LIN {X 0,Y 136.247,Z 303.137,A -85,B 0,C 180,E1 -24818.833,E2 -24818.833} C_VEL
LIN {X 0,Y 136.271,Z 303.129,A -85,B 0,C 180,E1 -24825.056,E2 -24825.056} C_VEL
LIN {X 0,Y 136.434,Z 303.114,A -85,B 0,C 180,E1 -24828.164,E2 -24828.164} C_VEL
LIN {X 0,Y 136.551,Z 303.099,A -85,B 0,C 180,E1 -24831.117,E2 -24831.117} C_VEL
LIN {X 0,Y 137.132,Z 303.026,A -85,B 0,C 180,E1 -24839.999,E2 -24839.999} C_VEL
LIN {X 0,Y 136.551,Z 303.097,A -85,B 0,C 180,E1 -24848.882,E2 -24848.882} C_VEL
LIN {X 0,Y 136.442,Z 303.112,A -85,B 0,C 180,E1 -24851.889,E2 -24851.889} C_VEL
LIN {X 0,Y 136.252,Z 303.133,A -85,B 0,C 180,E1 -24858.027,E2 -24858.027} C_VEL
LIN {X 0,Y 136.434,Z 303.14,A -85,B 0,C 180,E1 -24864.336,E2 -24864.336} C_VEL
LIN {X 0,Y 136.755,Z 306.874,A -85,B 0,C 180,E1 -24870.924,E2 -24870.924} C_VEL
LIN {X 0,Y 137.423,Z 309.535,A -85,B 0,C 180,E1 -24875.456,E2 -24875.456} C_VEL
LIN {X 0,Y 143.688,Z 330.399,A -85,B 0,C 180,E1 -24879.825,E2 -24879.825} C_VEL
LIN {X 0,Y 145.662,Z 339.16,A -85,B 0,C 180,E1 -24881.689,E2 -24881.689} C_VEL
LIN {X 0,Y 147.43,Z 355.491,A -85,B 0,C 180,E1 -24885.229,E2 -24885.229} C_VEL
LIN {X 0,Y 148.861,Z 369.384,A -85,B 0,C 180,E1 -24888.626,E2 -24888.626} C_VEL
LIN {X 0,Y 150.113,Z 381.659,A -85,B 0,C 180,E1 -24891.987,E2 -24891.987} C_VEL
LIN {X 0,Y 150.686,Z 388.239,A -85,B 0,C 180,E1 -24893.945,E2 -24893.945} C_VEL
LIN {X 0,Y 146.918,Z 399.34,A -85,B 0,C 180,E1 -24897.441,E2 -24897.441} C_VEL
LIN {X 0,Y 142.825,Z 411.303,A -85,B 0,C 180,E1 -24902.116,E2 -24902.116} C_VEL
LIN {X 0,Y 139.666,Z 421.52,A -85,B 0,C 180,E1 -24907.046,E2 -24907.046} C_VEL
LIN {X 0,Y 137.366,Z 430.082,A -85,B 0,C 180,E1 -24912.123,E2 -24912.123} C_VEL
LIN {X 0,Y 135.876,Z 438.21,A -85,B 0,C 180,E1 -24918.059,E2 -24918.059} C_VEL
LIN {X 0,Y 135.342,Z 444.688,A -85,B 0,C 180,E1 -24924.039,E2 -24924.039} C_VEL
LIN {X 0,Y 135.239,Z 448.491,A -85,B 0,C 180,E1 -24928.511,E2 -24928.511} C_VEL
LIN {X 0,Y 135.256,Z 449.575,A -85,B 0,C 180,E1 -24930,E2 -24930} C_VEL
LIN {X 0,Y 135.01,Z 451.418,A -85,B 0,C 180,E1 -24932.984,E2 -24932.984} C_VEL
LIN {X 0,Y 134.714,Z 453.637,A -85,B 0,C 180,E1 -24937.6,E2 -24937.6} C_VEL
LIN {X 0,Y 135.394,Z 456.033,A -85,B 0,C 180,E1 -24945.043,E2 -24945.043} C_VEL
LIN {X 0,Y 139.13,Z 457.397,A -85,B 0,C 180,E1 -24953.835,E2 -24953.835} C_VEL
LIN {X 0,Y 146.373,Z 457.366,A -85,B 0,C 180,E1 -24961.881,E2 -24961.881} C_VEL
LIN {X 0,Y 156.505,Z 456.017,A -85,B 0,C 180,E1 -24968.953,E2 -24968.953} C_VEL
LIN {X 0,Y 164.765,Z 454.523,A -85,B 0,C 180,E1 -24973.038,E2 -24973.038} C_VEL
LIN {X 0,Y 169.344,Z 453.57,A -85,B 0,C 180,E1 -24974.872,E2 -24974.872} C_VEL
LIN {X 0,Y 170.849,Z 453.204,A -85,B 0,C 180,E1 -24975.629,E2 -24975.629} C_VEL
LIN {X 0,Y 158.161,Z 452.885,A -85,B 0,C 180,E1 -24981.531,E2 -24981.531} C_VEL
LIN {X 0,Y 150.957,Z 451.853,A -85,B 0,C 180,E1 -24986.036,E2 -24986.036} C_VEL
LIN {X 0,Y 144.974,Z 450.016,A -85,B 0,C 180,E1 -24991.003,E2 -24991.003} C_VEL
LIN {X 0,Y 140.598,Z 447.636,A -85,B 0,C 180,E1 -24995.993,E2 -24995.993} C_VEL
LIN {X 0,Y 138.42,Z 446.349,A -85,B 0,C 180,E1 -24998.183,E2 -24998.183} C_VEL
LIN {X 0,Y 133.615,Z 443.7,A -85,B 0,C 180,E1 -25001.66,E2 -25001.66} C_VEL
LIN {X 0,Y 130.02,Z 441.226,A -85,B 0,C 180,E1 -25004.557,E2 -25004.557} C_VEL
LIN {X 0,Y 128.29,Z 439.216,A -85,B 0,C 180,E1 -25006.914,E2 -25006.914} C_VEL
LIN {X 0,Y 128.014,Z 438.527,A -85,B 0,C 180,E1 -25007.737,E2 -25007.737} C_VEL
LIN {X 0,Y 127.224,Z 432.975,A -85,B 0,C 180,E1 -25013.906,E2 -25013.906} C_VEL
LIN {X 0,Y 127.191,Z 428.154,A -85,B 0,C 180,E1 -25018.418,E2 -25018.418} C_VEL
LIN {X 0,Y 127.646,Z 420.139,A -85,B 0,C 180,E1 -25024.738,E2 -25024.738} C_VEL
LIN {X 0,Y 128.792,Z 410.762,A -85,B 0,C 180,E1 -25030.813,E2 -25030.813} C_VEL
LIN {X 0,Y 131.133,Z 398.794,A -85,B 0,C 180,E1 -25037.144,E2 -25037.144} C_VEL
LIN {X 0,Y 133.545,Z 388.569,A -85,B 0,C 180,E1 -25041.617,E2 -25041.617} C_VEL
LIN {X 0,Y 137.26,Z 374.549,A -85,B 0,C 180,E1 -25046.617,E2 -25046.617} C_VEL
LIN {X 0,Y 140.984,Z 360.329,A -85,B 0,C 180,E1 -25050.729,E2 -25050.729} C_VEL
LIN {X 0,Y 143.252,Z 351.164,A -85,B 0,C 180,E1 -25052.95,E2 -25052.95} C_VEL
LIN {X 0,Y 140.82,Z 340.487,A -85,B 0,C 180,E1 -25055.806,E2 -25055.806} C_VEL
LIN {X 0,Y 136.648,Z 326.02,A -85,B 0,C 180,E1 -25059.514,E2 -25059.514} C_VEL
LIN {X 0,Y 131.962,Z 312.426,A -85,B 0,C 180,E1 -25062.921,E2 -25062.921} C_VEL
LIN {X 0,Y 128.958,Z 304.05,A -85,B 0,C 180,E1 -25065.024,E2 -25065.024} C_VEL
LIN {X 0,Y 128.938,Z 304.048,A -85,B 0,C 180,E1 -25069.739,E2 -25069.739} C_VEL
LIN {X 0,Y 128.983,Z 304.045,A -85,B 0,C 180,E1 -25074.819,E2 -25074.819} C_VEL
LIN {X 0,Y 129.019,Z 304.038,A -85,B 0,C 180,E1 -25080.643,E2 -25080.643} C_VEL
LIN {X 0,Y 129.033,Z 304.037,A -85,B 0,C 180,E1 -25084.168,E2 -25084.168} C_VEL
LIN {X 0,Y 129.11,Z 304.023,A -85,B 0,C 180,E1 -25087.728,E2 -25087.728} C_VEL
LIN {X 0,Y 129.156,Z 304.021,A -85,B 0,C 180,E1 -25090.944,E2 -25090.944} C_VEL
LIN {X 0,Y 129.392,Z 303.991,A -85,B 0,C 180,E1 -25097.876,E2 -25097.876} C_VEL
LIN {X 0,Y 129.475,Z 303.98,A -85,B 0,C 180,E1 -25100.628,E2 -25100.628} C_VEL
LIN {X 0,Y 130.087,Z 303.902,A -85,B 0,C 180,E1 -25110,E2 -25110} C_VEL
LIN {X 0,Y 129.481,Z 303.976,A -85,B 0,C 180,E1 -25119.372,E2 -25119.372} C_VEL
LIN {X 0,Y 129.355,Z 303.996,A -85,B 0,C 180,E1 -25122.552,E2 -25122.552} C_VEL
LIN {X 0,Y 129.187,Z 304.013,A -85,B 0,C 180,E1 -25129.051,E2 -25129.051} C_VEL
LIN {X 0,Y 129.139,Z 304.023,A -85,B 0,C 180,E1 -25132.393,E2 -25132.393} C_VEL
LIN {X 0,Y 129.038,Z 304.037,A -85,B 0,C 180,E1 -25139.373,E2 -25139.373} C_VEL
LIN {X 0,Y 128.959,Z 304.041,A -85,B 0,C 180,E1 -25145.167,E2 -25145.167} C_VEL
LIN {X 0,Y 128.924,Z 304.048,A -85,B 0,C 180,E1 -25150.856,E2 -25150.856} C_VEL
LIN {X 0,Y 128.914,Z 304.052,A -85,B 0,C 180,E1 -25155.132,E2 -25155.132} C_VEL
LIN {X 0,Y 128.938,Z 304.044,A -85,B 0,C 180,E1 -25159.739,E2 -25159.739} C_VEL
LIN {X 0,Y 128.983,Z 304.044,A -85,B 0,C 180,E1 -25164.818,E2 -25164.818} C_VEL
LIN {X 0,Y 129.019,Z 304.036,A -85,B 0,C 180,E1 -25170.642,E2 -25170.642} C_VEL
LIN {X 0,Y 129.033,Z 304.037,A -85,B 0,C 180,E1 -25174.167,E2 -25174.167} C_VEL
LIN {X 0,Y 129.11,Z 304.021,A -85,B 0,C 180,E1 -25177.727,E2 -25177.727} C_VEL
LIN {X 0,Y 129.156,Z 304.022,A -85,B 0,C 180,E1 -25180.943,E2 -25180.943} C_VEL
LIN {X 0,Y 129.392,Z 303.99,A -85,B 0,C 180,E1 -25187.875,E2 -25187.875} C_VEL
LIN {X 0,Y 129.475,Z 303.981,A -85,B 0,C 180,E1 -25190.627,E2 -25190.627} C_VEL
LIN {X 0,Y 130.087,Z 303.904,A -85,B 0,C 180,E1 -25199.999,E2 -25199.999} C_VEL
LIN {X 0,Y 129.477,Z 303.978,A -85,B 0,C 180,E1 -25209.371,E2 -25209.371} C_VEL
LIN {X 0,Y 129.346,Z 303.996,A -85,B 0,C 180,E1 -25212.552,E2 -25212.552} C_VEL
LIN {X 0,Y 129.179,Z 304.015,A -85,B 0,C 180,E1 -25219.052,E2 -25219.052} C_VEL
LIN {X 0,Y 129.367,Z 304.154,A -85,B 0,C 180,E1 -25224.898,E2 -25224.898} C_VEL
LIN {X 0,Y 129.882,Z 308.439,A -85,B 0,C 180,E1 -25232.758,E2 -25232.758} C_VEL
LIN {X 0,Y 130.109,Z 309.14,A -85,B 0,C 180,E1 -25233.967,E2 -25233.967} C_VEL
LIN {X 0,Y 136.026,Z 328.806,A -85,B 0,C 180,E1 -25238.315,E2 -25238.315} C_VEL
LIN {X 0,Y 138.682,Z 339.25,A -85,B 0,C 180,E1 -25240.718,E2 -25240.718} C_VEL
LIN {X 0,Y 140.292,Z 353.804,A -85,B 0,C 180,E1 -25244.032,E2 -25244.032} C_VEL
LIN {X 0,Y 141.788,Z 369.4,A -85,B 0,C 180,E1 -25248.03,E2 -25248.03} C_VEL
LIN {X 0,Y 143.073,Z 382.421,A -85,B 0,C 180,E1 -25251.807,E2 -25251.807} C_VEL
LIN {X 0,Y 143.609,Z 387.897,A -85,B 0,C 180,E1 -25253.526,E2 -25253.526} C_VEL
LIN {X 0,Y 139.712,Z 399.089,A -85,B 0,C 180,E1 -25257.264,E2 -25257.264} C_VEL
LIN {X 0,Y 135.93,Z 409.933,A -85,B 0,C 180,E1 -25261.706,E2 -25261.706} C_VEL
LIN {X 0,Y 132.843,Z 419.722,A -85,B 0,C 180,E1 -25266.622,E2 -25266.622} C_VEL
LIN {X 0,Y 130.472,Z 428.371,A -85,B 0,C 180,E1 -25271.957,E2 -25271.957} C_VEL
LIN {X 0,Y 129.087,Z 435.667,A -85,B 0,C 180,E1 -25277.421,E2 -25277.421} C_VEL
LIN {X 0,Y 128.494,Z 442.455,A -85,B 0,C 180,E1 -25283.72,E2 -25283.72} C_VEL
LIN {X 0,Y 128.382,Z 446.483,A -85,B 0,C 180,E1 -25288.431,E2 -25288.431} C_VEL
LIN {X 0,Y 128.387,Z 447.654,A -85,B 0,C 180,E1 -25290,E2 -25290} C_VEL
LIN {X 0,Y 128.146,Z 449.612,A -85,B 0,C 180,E1 -25293.144,E2 -25293.144} C_VEL
LIN {X 0,Y 127.839,Z 452.095,A -85,B 0,C 180,E1 -25298.294,E2 -25298.294} C_VEL
LIN {X 0,Y 128.636,Z 454.561,A -85,B 0,C 180,E1 -25305.853,E2 -25305.853} C_VEL
LIN {X 0,Y 132.681,Z 456.227,A -85,B 0,C 180,E1 -25315.072,E2 -25315.072} C_VEL
LIN {X 0,Y 140.385,Z 456.546,A -85,B 0,C 180,E1 -25323.414,E2 -25323.414} C_VEL
LIN {X 0,Y 151.043,Z 455.659,A -85,B 0,C 180,E1 -25330.649,E2 -25330.649} C_VEL
LIN {X 0,Y 159.649,Z 454.433,A -85,B 0,C 180,E1 -25334.777,E2 -25334.777} C_VEL
LIN {X 0,Y 161.243,Z 454.077,A -85,B 0,C 180,E1 -25335.783,E2 -25335.783} C_VEL
LIN {X 0,Y 152.661,Z 453.441,A -85,B 0,C 180,E1 -25339.872,E2 -25339.872} C_VEL
LIN {X 0,Y 141.781,Z 451.137,A -85,B 0,C 180,E1 -25346.958,E2 -25346.958} C_VEL
LIN {X 0,Y 136.124,Z 448.673,A -85,B 0,C 180,E1 -25352.312,E2 -25352.312} C_VEL
LIN {X 0,Y 131.776,Z 445.435,A -85,B 0,C 180,E1 -25358.08,E2 -25358.08} C_VEL
LIN {X 0,Y 128.491,Z 440.128,A -85,B 0,C 180,E1 -25365.752,E2 -25365.752} C_VEL
LIN {X 0,Y 128.014,Z 438.527,A -85,B 0,C 180,E1 -25367.737,E2 -25367.737} C_VEL
LIN {X 0,Y 126.912,Z 436.36,A -85,B 0,C 180,E1 -25370.152,E2 -25370.152} C_VEL
LIN {X 0,Y 125.08,Z 433.957,A -85,B 0,C 180,E1 -25372.473,E2 -25372.473} C_VEL
LIN {X 0,Y 121.241,Z 428.484,A -85,B 0,C 180,E1 -25377.122,E2 -25377.122} C_VEL
LIN {X 0,Y 120.269,Z 425.573,A -85,B 0,C 180,E1 -25379.558,E2 -25379.558} C_VEL
LIN {X 0,Y 120.223,Z 424.572,A -85,B 0,C 180,E1 -25380.384,E2 -25380.384} C_VEL
LIN {X 0,Y 120.757,Z 417.504,A -85,B 0,C 180,E1 -25385.846,E2 -25385.846} C_VEL
LIN {X 0,Y 122.135,Z 407.431,A -85,B 0,C 180,E1 -25392.378,E2 -25392.378} C_VEL
LIN {X 0,Y 124.432,Z 396.651,A -85,B 0,C 180,E1 -25398.099,E2 -25398.099} C_VEL
LIN {X 0,Y 127.486,Z 384.124,A -85,B 0,C 180,E1 -25403.559,E2 -25403.559} C_VEL
LIN {X 0,Y 130.911,Z 371.667,A -85,B 0,C 180,E1 -25408.019,E2 -25408.019} C_VEL
LIN {X 0,Y 134.564,Z 358.197,A -85,B 0,C 180,E1 -25411.921,E2 -25411.921} C_VEL
LIN {X 0,Y 136.065,Z 352.541,A -85,B 0,C 180,E1 -25413.345,E2 -25413.345} C_VEL
LIN {X 0,Y 135.805,Z 349.78,A -85,B 0,C 180,E1 -25414.104,E2 -25414.104} C_VEL
LIN {X 0,Y 132.825,Z 337.831,A -85,B 0,C 180,E1 -25417.469,E2 -25417.469} C_VEL
LIN {X 0,Y 128.684,Z 324.087,A -85,B 0,C 180,E1 -25421.208,E2 -25421.208} C_VEL
LIN {X 0,Y 123.585,Z 309.815,A -85,B 0,C 180,E1 -25424.977,E2 -25424.977} C_VEL
LIN {X 0,Y 121.846,Z 304.934,A -85,B 0,C 180,E1 -25426.367,E2 -25426.367} C_VEL
LIN {X 0,Y 121.858,Z 304.931,A -85,B 0,C 180,E1 -25430.623,E2 -25430.623} C_VEL
LIN {X 0,Y 121.935,Z 304.922,A -85,B 0,C 180,E1 -25434.804,E2 -25434.804} C_VEL
LIN {X 0,Y 121.931,Z 304.921,A -85,B 0,C 180,E1 -25439.837,E2 -25439.837} C_VEL
LIN {X 0,Y 121.986,Z 304.909,A -85,B 0,C 180,E1 -25446.216,E2 -25446.216} C_VEL
LIN {X 0,Y 122.048,Z 304.906,A -85,B 0,C 180,E1 -25449.787,E2 -25449.787} C_VEL
LIN {X 0,Y 122.242,Z 304.882,A -85,B 0,C 180,E1 -25456.705,E2 -25456.705} C_VEL
LIN {X 0,Y 122.411,Z 304.862,A -85,B 0,C 180,E1 -25460.082,E2 -25460.082} C_VEL
LIN {X 0,Y 122.591,Z 304.839,A -85,B 0,C 180,E1 -25466.714,E2 -25466.714} C_VEL
LIN {X 0,Y 123.04,Z 304.779,A -85,B 0,C 180,E1 -25470,E2 -25470} C_VEL
LIN {X 0,Y 122.424,Z 304.859,A -85,B 0,C 180,E1 -25476.593,E2 -25476.593} C_VEL
LIN {X 0,Y 122.417,Z 304.856,A -85,B 0,C 180,E1 -25479.918,E2 -25479.918} C_VEL
LIN {X 0,Y 122.249,Z 304.882,A -85,B 0,C 180,E1 -25483.295,E2 -25483.295} C_VEL
LIN {X 0,Y 122.076,Z 304.903,A -85,B 0,C 180,E1 -25490.208,E2 -25490.208} C_VEL
LIN {X 0,Y 121.999,Z 304.911,A -85,B 0,C 180,E1 -25493.782,E2 -25493.782} C_VEL
LIN {X 0,Y 121.942,Z 304.92,A -85,B 0,C 180,E1 -25500.171,E2 -25500.171} C_VEL
LIN {X 0,Y 121.883,Z 304.925,A -85,B 0,C 180,E1 -25506.169,E2 -25506.169} C_VEL
LIN {X 0,Y 121.865,Z 304.925,A -85,B 0,C 180,E1 -25511.433,E2 -25511.433} C_VEL
LIN {X 0,Y 121.866,Z 304.929,A -85,B 0,C 180,E1 -25518.566,E2 -25518.566} C_VEL
LIN {X 0,Y 121.935,Z 304.922,A -85,B 0,C 180,E1 -25524.803,E2 -25524.803} C_VEL
LIN {X 0,Y 121.931,Z 304.916,A -85,B 0,C 180,E1 -25529.836,E2 -25529.836} C_VEL
LIN {X 0,Y 121.986,Z 304.91,A -85,B 0,C 180,E1 -25536.215,E2 -25536.215} C_VEL
LIN {X 0,Y 122.048,Z 304.905,A -85,B 0,C 180,E1 -25539.787,E2 -25539.787} C_VEL
LIN {X 0,Y 122.242,Z 304.879,A -85,B 0,C 180,E1 -25546.704,E2 -25546.704} C_VEL
LIN {X 0,Y 122.411,Z 304.863,A -85,B 0,C 180,E1 -25550.081,E2 -25550.081} C_VEL
LIN {X 0,Y 122.594,Z 304.839,A -85,B 0,C 180,E1 -25556.713,E2 -25556.713} C_VEL
LIN {X 0,Y 123.041,Z 304.781,A -85,B 0,C 180,E1 -25559.999,E2 -25559.999} C_VEL
LIN {X 0,Y 122.423,Z 304.86,A -85,B 0,C 180,E1 -25566.592,E2 -25566.592} C_VEL
LIN {X 0,Y 122.407,Z 304.857,A -85,B 0,C 180,E1 -25569.918,E2 -25569.918} C_VEL
LIN {X 0,Y 122.242,Z 304.882,A -85,B 0,C 180,E1 -25573.295,E2 -25573.295} C_VEL
LIN {X 0,Y 122.118,Z 304.899,A -85,B 0,C 180,E1 -25580.2,E2 -25580.2} C_VEL
LIN {X 0,Y 122.314,Z 304.914,A -85,B 0,C 180,E1 -25585.071,E2 -25585.071} C_VEL
LIN {X 0,Y 122.754,Z 308.868,A -85,B 0,C 180,E1 -25592.34,E2 -25592.34} C_VEL
LIN {X 0,Y 127.805,Z 325.454,A -85,B 0,C 180,E1 -25596.272,E2 -25596.272} C_VEL
LIN {X 0,Y 131.407,Z 338.28,A -85,B 0,C 180,E1 -25599.427,E2 -25599.427} C_VEL
LIN {X 0,Y 132.448,Z 344.471,A -85,B 0,C 180,E1 -25600.907,E2 -25600.907} C_VEL
LIN {X 0,Y 133.798,Z 359.38,A -85,B 0,C 180,E1 -25604.631,E2 -25604.631} C_VEL
LIN {X 0,Y 135.224,Z 374.386,A -85,B 0,C 180,E1 -25608.901,E2 -25608.901} C_VEL
LIN {X 0,Y 136.456,Z 387.871,A -85,B 0,C 180,E1 -25613.221,E2 -25613.221} C_VEL
LIN {X 0,Y 131.894,Z 400.51,A -85,B 0,C 180,E1 -25617.801,E2 -25617.801} C_VEL
LIN {X 0,Y 127.911,Z 412.021,A -85,B 0,C 180,E1 -25623.045,E2 -25623.045} C_VEL
LIN {X 0,Y 124.607,Z 423.026,A -85,B 0,C 180,E1 -25629.359,E2 -25629.359} C_VEL
LIN {X 0,Y 122.525,Z 432.013,A -85,B 0,C 180,E1 -25635.89,E2 -25635.89} C_VEL
LIN {X 0,Y 121.753,Z 438.493,A -85,B 0,C 180,E1 -25641.703,E2 -25641.703} C_VEL
LIN {X 0,Y 121.596,Z 443.062,A -85,B 0,C 180,E1 -25646.686,E2 -25646.686} C_VEL
LIN {X 0,Y 121.575,Z 445.568,A -85,B 0,C 180,E1 -25650,E2 -25650} C_VEL
LIN {X 0,Y 121.339,Z 447.639,A -85,B 0,C 180,E1 -25653.32,E2 -25653.32} C_VEL
LIN {X 0,Y 121.022,Z 450.427,A -85,B 0,C 180,E1 -25659.174,E2 -25659.174} C_VEL
LIN {X 0,Y 121.921,Z 452.992,A -85,B 0,C 180,E1 -25666.751,E2 -25666.751} C_VEL
LIN {X 0,Y 126.339,Z 454.977,A -85,B 0,C 180,E1 -25676.425,E2 -25676.425} C_VEL
LIN {X 0,Y 134.514,Z 455.608,A -85,B 0,C 180,E1 -25685.08,E2 -25685.08} C_VEL
LIN {X 0,Y 145.726,Z 455.082,A -85,B 0,C 180,E1 -25692.469,E2 -25692.469} C_VEL
LIN {X 0,Y 150.039,Z 454.695,A -85,B 0,C 180,E1 -25694.638,E2 -25694.638} C_VEL
LIN {X 0,Y 151.661,Z 454.387,A -85,B 0,C 180,E1 -25695.965,E2 -25695.965} C_VEL
LIN {X 0,Y 139.375,Z 452.212,A -85,B 0,C 180,E1 -25702.765,E2 -25702.765} C_VEL
LIN {X 0,Y 129.857,Z 448.425,A -85,B 0,C 180,E1 -25710.851,E2 -25710.851} C_VEL
LIN {X 0,Y 124.324,Z 443.944,A -85,B 0,C 180,E1 -25718.443,E2 -25718.443} C_VEL
LIN {X 0,Y 121.217,Z 438.065,A -85,B 0,C 180,E1 -25726.591,E2 -25726.591} C_VEL
LIN {X 0,Y 120.196,Z 431.125,A -85,B 0,C 180,E1 -25734.391,E2 -25734.391} C_VEL
LIN {X 0,Y 120.223,Z 424.572,A -85,B 0,C 180,E1 -25740.384,E2 -25740.384} C_VEL
LIN {X 0,Y 119.727,Z 421.513,A -85,B 0,C 180,E1 -25742.772,E2 -25742.772} C_VEL
LIN {X 0,Y 117.359,Z 415.925,A -85,B 0,C 180,E1 -25746.56,E2 -25746.56} C_VEL
LIN {X 0,Y 115.233,Z 409.915,A -85,B 0,C 180,E1 -25750.363,E2 -25750.363} C_VEL
LIN {X 0,Y 115.169,Z 406.133,A -85,B 0,C 180,E1 -25752.676,E2 -25752.676} C_VEL
LIN {X 0,Y 117.766,Z 394.384,A -85,B 0,C 180,E1 -25759.162,E2 -25759.162} C_VEL
LIN {X 0,Y 121.105,Z 381.441,A -85,B 0,C 180,E1 -25764.882,E2 -25764.882} C_VEL
LIN {X 0,Y 124.724,Z 368.482,A -85,B 0,C 180,E1 -25769.542,E2 -25769.542} C_VEL
LIN {X 0,Y 128.634,Z 354.502,A -85,B 0,C 180,E1 -25773.635,E2 -25773.635} C_VEL
LIN {X 0,Y 129.041,Z 352.938,A -85,B 0,C 180,E1 -25774.032,E2 -25774.032} C_VEL
LIN {X 0,Y 128.281,Z 348.307,A -85,B 0,C 180,E1 -25775.419,E2 -25775.419} C_VEL
LIN {X 0,Y 125.012,Z 336.071,A -85,B 0,C 180,E1 -25779.024,E2 -25779.024} C_VEL
LIN {X 0,Y 121.156,Z 323.601,A -85,B 0,C 180,E1 -25782.602,E2 -25782.602} C_VEL
LIN {X 0,Y 115.826,Z 308.712,A -85,B 0,C 180,E1 -25786.873,E2 -25786.873} C_VEL
LIN {X 0,Y 114.806,Z 305.807,A -85,B 0,C 180,E1 -25787.82,E2 -25787.82} C_VEL
LIN {X 0,Y 114.798,Z 305.81,A -85,B 0,C 180,E1 -25792.739,E2 -25792.739} C_VEL
LIN {X 0,Y 114.865,Z 305.802,A -85,B 0,C 180,E1 -25798.938,E2 -25798.938} C_VEL
LIN {X 0,Y 114.95,Z 305.785,A -85,B 0,C 180,E1 -25806.507,E2 -25806.507} C_VEL
LIN {X 0,Y 115.014,Z 305.783,A -85,B 0,C 180,E1 -25812.21,E2 -25812.21} C_VEL
LIN {X 0,Y 115.252,Z 305.752,A -85,B 0,C 180,E1 -25817.341,E2 -25817.341} C_VEL
LIN {X 0,Y 115.361,Z 305.733,A -85,B 0,C 180,E1 -25823.002,E2 -25823.002} C_VEL
LIN {X 0,Y 115.992,Z 305.657,A -85,B 0,C 180,E1 -25830,E2 -25830} C_VEL
LIN {X 0,Y 115.366,Z 305.738,A -85,B 0,C 180,E1 -25836.998,E2 -25836.998} C_VEL
LIN {X 0,Y 115.256,Z 305.752,A -85,B 0,C 180,E1 -25842.669,E2 -25842.669} C_VEL
LIN {X 0,Y 115.034,Z 305.775,A -85,B 0,C 180,E1 -25847.787,E2 -25847.787} C_VEL
LIN {X 0,Y 114.969,Z 305.788,A -85,B 0,C 180,E1 -25853.514,E2 -25853.514} C_VEL
LIN {X 0,Y 114.864,Z 305.803,A -85,B 0,C 180,E1 -25861.061,E2 -25861.061} C_VEL
LIN {X 0,Y 114.777,Z 305.813,A -85,B 0,C 180,E1 -25867.758,E2 -25867.758} C_VEL
LIN {X 0,Y 114.78,Z 305.806,A -85,B 0,C 180,E1 -25872.711,E2 -25872.711} C_VEL
LIN {X 0,Y 114.789,Z 305.81,A -85,B 0,C 180,E1 -25877.663,E2 -25877.663} C_VEL
LIN {X 0,Y 114.798,Z 305.808,A -85,B 0,C 180,E1 -25882.738,E2 -25882.738} C_VEL
LIN {X 0,Y 114.865,Z 305.796,A -85,B 0,C 180,E1 -25888.937,E2 -25888.937} C_VEL
LIN {X 0,Y 114.95,Z 305.785,A -85,B 0,C 180,E1 -25896.506,E2 -25896.506} C_VEL
LIN {X 0,Y 115.014,Z 305.784,A -85,B 0,C 180,E1 -25902.209,E2 -25902.209} C_VEL
LIN {X 0,Y 115.251,Z 305.751,A -85,B 0,C 180,E1 -25907.34,E2 -25907.34} C_VEL
LIN {X 0,Y 115.363,Z 305.734,A -85,B 0,C 180,E1 -25913.001,E2 -25913.001} C_VEL
LIN {X 0,Y 115.992,Z 305.659,A -85,B 0,C 180,E1 -25919.999,E2 -25919.999} C_VEL
LIN {X 0,Y 115.364,Z 305.739,A -85,B 0,C 180,E1 -25926.997,E2 -25926.997} C_VEL
LIN {X 0,Y 115.248,Z 305.753,A -85,B 0,C 180,E1 -25932.653,E2 -25932.653} C_VEL
LIN {X 0,Y 115.04,Z 305.775,A -85,B 0,C 180,E1 -25937.785,E2 -25937.785} C_VEL
LIN {X 0,Y 115.275,Z 305.752,A -85,B 0,C 180,E1 -25943.863,E2 -25943.863} C_VEL
LIN {X 0,Y 115.249,Z 305.863,A -85,B 0,C 180,E1 -25945.752,E2 -25945.752} C_VEL
LIN {X 0,Y 115.46,Z 308.273,A -85,B 0,C 180,E1 -25950.532,E2 -25950.532} C_VEL
LIN {X 0,Y 120.435,Z 324.536,A -85,B 0,C 180,E1 -25954.677,E2 -25954.677} C_VEL
LIN {X 0,Y 124.741,Z 340.244,A -85,B 0,C 180,E1 -25958.813,E2 -25958.813} C_VEL
LIN {X 0,Y 125.727,Z 346.936,A -85,B 0,C 180,E1 -25960.527,E2 -25960.527} C_VEL
LIN {X 0,Y 127.092,Z 362.855,A -85,B 0,C 180,E1 -25964.86,E2 -25964.86} C_VEL
LIN {X 0,Y 128.455,Z 378.09,A -85,B 0,C 180,E1 -25969.566,E2 -25969.566} C_VEL
LIN {X 0,Y 129.284,Z 387.429,A -85,B 0,C 180,E1 -25972.788,E2 -25972.788} C_VEL
LIN {X 0,Y 125.301,Z 398.399,A -85,B 0,C 180,E1 -25976.949,E2 -25976.949} C_VEL
LIN {X 0,Y 121.221,Z 409.913,A -85,B 0,C 180,E1 -25982.366,E2 -25982.366} C_VEL
LIN {X 0,Y 118.129,Z 419.782,A -85,B 0,C 180,E1 -25988.171,E2 -25988.171} C_VEL
LIN {X 0,Y 115.844,Z 429.158,A -85,B 0,C 180,E1 -25995.058,E2 -25995.058} C_VEL
LIN {X 0,Y 114.95,Z 435.953,A -85,B 0,C 180,E1 -26001.208,E2 -26001.208} C_VEL
LIN {X 0,Y 114.789,Z 440.725,A -85,B 0,C 180,E1 -26006.49,E2 -26006.49} C_VEL
LIN {X 0,Y 114.774,Z 443.406,A -85,B 0,C 180,E1 -26010,E2 -26010} C_VEL
LIN {X 0,Y 114.564,Z 445.565,A -85,B 0,C 180,E1 -26013.517,E2 -26013.517} C_VEL
LIN {X 0,Y 114.235,Z 448.689,A -85,B 0,C 180,E1 -26020.152,E2 -26020.152} C_VEL
LIN {X 0,Y 115.298,Z 451.236,A -85,B 0,C 180,E1 -26027.745,E2 -26027.745} C_VEL
LIN {X 0,Y 120.087,Z 453.517,A -85,B 0,C 180,E1 -26037.917,E2 -26037.917} C_VEL
LIN {X 0,Y 128.793,Z 454.544,A -85,B 0,C 180,E1 -26046.888,E2 -26046.888} C_VEL
LIN {X 0,Y 140.569,Z 454.362,A -85,B 0,C 180,E1 -26054.424,E2 -26054.424} C_VEL
LIN {X 0,Y 142.101,Z 454.058,A -85,B 0,C 180,E1 -26056.18,E2 -26056.18} C_VEL
LIN {X 0,Y 130.06,Z 450.965,A -85,B 0,C 180,E1 -26063.531,E2 -26063.531} C_VEL
LIN {X 0,Y 123.687,Z 448.019,A -85,B 0,C 180,E1 -26069.245,E2 -26069.245} C_VEL
LIN {X 0,Y 117.746,Z 443.227,A -85,B 0,C 180,E1 -26077.173,E2 -26077.173} C_VEL
LIN {X 0,Y 114.388,Z 437.077,A -85,B 0,C 180,E1 -26085.774,E2 -26085.774} C_VEL
LIN {X 0,Y 113.323,Z 431.022,A -85,B 0,C 180,E1 -26092.876,E2 -26092.876} C_VEL
LIN {X 0,Y 113.216,Z 425.602,A -85,B 0,C 180,E1 -26098.222,E2 -26098.222} C_VEL
LIN {X 0,Y 113.698,Z 417.057,A -85,B 0,C 180,E1 -26105.321,E2 -26105.321} C_VEL
LIN {X 0,Y 115.022,Z 407.003,A -85,B 0,C 180,E1 -26112.143,E2 -26112.143} C_VEL
LIN {X 0,Y 115.169,Z 406.133,A -85,B 0,C 180,E1 -26112.676,E2 -26112.676} C_VEL
LIN {X 0,Y 115.233,Z 402.313,A -85,B 0,C 180,E1 -26114.906,E2 -26114.906} C_VEL
LIN {X 0,Y 113.849,Z 395.57,A -85,B 0,C 180,E1 -26118.479,E2 -26118.479} C_VEL
LIN {X 0,Y 112.723,Z 388.498,A -85,B 0,C 180,E1 -26121.986,E2 -26121.986} C_VEL
LIN {X 0,Y 113.208,Z 384.083,A -85,B 0,C 180,E1 -26124.015,E2 -26124.015} C_VEL
LIN {X 0,Y 116.987,Z 370.956,A -85,B 0,C 180,E1 -26129.218,E2 -26129.218} C_VEL
LIN {X 0,Y 120.859,Z 357.45,A -85,B 0,C 180,E1 -26133.535,E2 -26133.535} C_VEL
LIN {X 0,Y 122.052,Z 352.998,A -85,B 0,C 180,E1 -26134.78,E2 -26134.78} C_VEL
LIN {X 0,Y 119.533,Z 342.507,A -85,B 0,C 180,E1 -26138.15,E2 -26138.15} C_VEL
LIN {X 0,Y 115.845,Z 329.766,A -85,B 0,C 180,E1 -26142.126,E2 -26142.126} C_VEL
LIN {X 0,Y 111.504,Z 316.881,A -85,B 0,C 180,E1 -26146.106,E2 -26146.106} C_VEL
LIN {X 0,Y 107.787,Z 306.684,A -85,B 0,C 180,E1 -26149.305,E2 -26149.305} C_VEL
LIN {X 0,Y 107.725,Z 306.691,A -85,B 0,C 180,E1 -26154.044,E2 -26154.044} C_VEL
LIN {X 0,Y 107.803,Z 306.683,A -85,B 0,C 180,E1 -26158.564,E2 -26158.564} C_VEL
LIN {X 0,Y 107.914,Z 306.662,A -85,B 0,C 180,E1 -26166.999,E2 -26166.999} C_VEL
LIN {X 0,Y 108.033,Z 306.646,A -85,B 0,C 180,E1 -26174.917,E2 -26174.917} C_VEL
LIN {X 0,Y 108.255,Z 306.625,A -85,B 0,C 180,E1 -26178.769,E2 -26178.769} C_VEL
LIN {X 0,Y 108.44,Z 306.603,A -85,B 0,C 180,E1 -26186.284,E2 -26186.284} C_VEL
LIN {X 0,Y 108.917,Z 306.538,A -85,B 0,C 180,E1 -26190,E2 -26190} C_VEL
LIN {X 0,Y 108.306,Z 306.617,A -85,B 0,C 180,E1 -26197.457,E2 -26197.457} C_VEL
LIN {X 0,Y 108.177,Z 306.634,A -85,B 0,C 180,E1 -26202.959,E2 -26202.959} C_VEL
LIN {X 0,Y 107.93,Z 306.661,A -85,B 0,C 180,E1 -26209.001,E2 -26209.001} C_VEL
LIN {X 0,Y 107.875,Z 306.669,A -85,B 0,C 180,E1 -26214.201,E2 -26214.201} C_VEL
LIN {X 0,Y 107.785,Z 306.681,A -85,B 0,C 180,E1 -26222.041,E2 -26222.041} C_VEL
LIN {X 0,Y 107.686,Z 306.696,A -85,B 0,C 180,E1 -26228.447,E2 -26228.447} C_VEL
LIN {X 0,Y 107.672,Z 306.697,A -85,B 0,C 180,E1 -26235.89,E2 -26235.89} C_VEL
LIN {X 0,Y 107.693,Z 306.69,A -85,B 0,C 180,E1 -26241.547,E2 -26241.547} C_VEL
LIN {X 0,Y 107.803,Z 306.675,A -85,B 0,C 180,E1 -26248.563,E2 -26248.563} C_VEL
LIN {X 0,Y 107.914,Z 306.661,A -85,B 0,C 180,E1 -26256.998,E2 -26256.998} C_VEL
LIN {X 0,Y 108.033,Z 306.646,A -85,B 0,C 180,E1 -26264.916,E2 -26264.916} C_VEL
LIN {X 0,Y 108.254,Z 306.625,A -85,B 0,C 180,E1 -26268.768,E2 -26268.768} C_VEL
LIN {X 0,Y 108.442,Z 306.601,A -85,B 0,C 180,E1 -26276.283,E2 -26276.283} C_VEL
LIN {X 0,Y 108.918,Z 306.54,A -85,B 0,C 180,E1 -26279.999,E2 -26279.999} C_VEL
LIN {X 0,Y 108.303,Z 306.619,A -85,B 0,C 180,E1 -26287.456,E2 -26287.456} C_VEL
LIN {X 0,Y 108.17,Z 306.634,A -85,B 0,C 180,E1 -26292.945,E2 -26292.945} C_VEL
LIN {X 0,Y 107.967,Z 306.656,A -85,B 0,C 180,E1 -26298.993,E2 -26298.993} C_VEL
LIN {X 0,Y 108.216,Z 306.632,A -85,B 0,C 180,E1 -26305.477,E2 -26305.477} C_VEL
LIN {X 0,Y 108.193,Z 307.022,A -85,B 0,C 180,E1 -26307.045,E2 -26307.045} C_VEL
LIN {X 0,Y 108.236,Z 307.9,A -85,B 0,C 180,E1 -26308.611,E2 -26308.611} C_VEL
LIN {X 0,Y 109.953,Z 313.841,A -85,B 0,C 180,E1 -26310.221,E2 -26310.221} C_VEL
LIN {X 0,Y 114.159,Z 327.594,A -85,B 0,C 180,E1 -26314.044,E2 -26314.044} C_VEL
LIN {X 0,Y 118.137,Z 342.545,A -85,B 0,C 180,E1 -26318.278,E2 -26318.278} C_VEL
LIN {X 0,Y 119.068,Z 350.537,A -85,B 0,C 180,E1 -26320.486,E2 -26320.486} C_VEL
LIN {X 0,Y 120.284,Z 365.797,A -85,B 0,C 180,E1 -26325.026,E2 -26325.026} C_VEL
LIN {X 0,Y 121.509,Z 379.802,A -85,B 0,C 180,E1 -26329.724,E2 -26329.724} C_VEL
LIN {X 0,Y 122.096,Z 386.794,A -85,B 0,C 180,E1 -26332.295,E2 -26332.295} C_VEL
LIN {X 0,Y 120.357,Z 391.975,A -85,B 0,C 180,E1 -26334.272,E2 -26334.272} C_VEL
LIN {X 0,Y 115.685,Z 404.417,A -85,B 0,C 180,E1 -26339.92,E2 -26339.92} C_VEL
LIN {X 0,Y 112.152,Z 414.968,A -85,B 0,C 180,E1 -26345.963,E2 -26345.963} C_VEL
LIN {X 0,Y 109.712,Z 423.874,A -85,B 0,C 180,E1 -26352.285,E2 -26352.285} C_VEL
LIN {X 0,Y 108.388,Z 431.321,A -85,B 0,C 180,E1 -26358.783,E2 -26358.783} C_VEL
LIN {X 0,Y 108.042,Z 436.681,A -85,B 0,C 180,E1 -26364.4,E2 -26364.4} C_VEL
LIN {X 0,Y 108.032,Z 441.038,A -85,B 0,C 180,E1 -26370,E2 -26370} C_VEL
LIN {X 0,Y 107.846,Z 443.343,A -85,B 0,C 180,E1 -26373.736,E2 -26373.736} C_VEL
LIN {X 0,Y 107.596,Z 445.261,A -85,B 0,C 180,E1 -26377.506,E2 -26377.506} C_VEL
LIN {X 0,Y 108.737,Z 449.392,A -85,B 0,C 180,E1 -26388.855,E2 -26388.855} C_VEL
LIN {X 0,Y 113.961,Z 451.929,A -85,B 0,C 180,E1 -26399.562,E2 -26399.562} C_VEL
LIN {X 0,Y 123.243,Z 453.257,A -85,B 0,C 180,E1 -26408.85,E2 -26408.85} C_VEL
LIN {X 0,Y 132.602,Z 453.497,A -85,B 0,C 180,E1 -26414.964,E2 -26414.964} C_VEL
LIN {X 0,Y 133.327,Z 453.342,A -85,B 0,C 180,E1 -26416.014,E2 -26416.014} C_VEL
LIN {X 0,Y 124.417,Z 450.688,A -85,B 0,C 180,E1 -26421.585,E2 -26421.585} C_VEL
LIN {X 0,Y 114.812,Z 445.645,A -85,B 0,C 180,E1 -26430.68,E2 -26430.68} C_VEL
LIN {X 0,Y 109.499,Z 440.04,A -85,B 0,C 180,E1 -26439.33,E2 -26439.33} C_VEL
LIN {X 0,Y 106.859,Z 433.003,A -85,B 0,C 180,E1 -26448.621,E2 -26448.621} C_VEL
LIN {X 0,Y 106.263,Z 426.065,A -85,B 0,C 180,E1 -26456.209,E2 -26456.209} C_VEL
LIN {X 0,Y 106.574,Z 417.664,A -85,B 0,C 180,E1 -26463.782,E2 -26463.782} C_VEL
LIN {X 0,Y 107.808,Z 407.485,A -85,B 0,C 180,E1 -26471.279,E2 -26471.279} C_VEL
LIN {X 0,Y 110.343,Z 395.238,A -85,B 0,C 180,E1 -26478.571,E2 -26478.571} C_VEL
LIN {X 0,Y 113.208,Z 384.083,A -85,B 0,C 180,E1 -26484.015,E2 -26484.015} C_VEL
LIN {X 0,Y 113.77,Z 379.652,A -85,B 0,C 180,E1 -26485.953,E2 -26485.953} C_VEL
LIN {X 0,Y 113.156,Z 371.981,A -85,B 0,C 180,E1 -26489.121,E2 -26489.121} C_VEL
LIN {X 0,Y 112.674,Z 364.072,A -85,B 0,C 180,E1 -26492.159,E2 -26492.159} C_VEL
LIN {X 0,Y 113.427,Z 359.141,A -85,B 0,C 180,E1 -26493.808,E2 -26493.808} C_VEL
LIN {X 0,Y 114.864,Z 354.038,A -85,B 0,C 180,E1 -26495.338,E2 -26495.338} C_VEL
LIN {X 0,Y 113.777,Z 348.407,A -85,B 0,C 180,E1 -26497.275,E2 -26497.275} C_VEL
LIN {X 0,Y 110.028,Z 334.63,A -85,B 0,C 180,E1 -26501.914,E2 -26501.914} C_VEL
LIN {X 0,Y 105.213,Z 319.907,A -85,B 0,C 180,E1 -26506.789,E2 -26506.789} C_VEL
LIN {X 0,Y 100.711,Z 307.565,A -85,B 0,C 180,E1 -26511.093,E2 -26511.093} C_VEL
LIN {X 0,Y 100.697,Z 307.567,A -85,B 0,C 180,E1 -26516.882,E2 -26516.882} C_VEL
LIN {X 0,Y 100.788,Z 307.551,A -85,B 0,C 180,E1 -26525.268,E2 -26525.268} C_VEL
LIN {X 0,Y 100.819,Z 307.551,A -85,B 0,C 180,E1 -26529.602,E2 -26529.602} C_VEL
LIN {X 0,Y 101.103,Z 307.514,A -85,B 0,C 180,E1 -26536.707,E2 -26536.707} C_VEL
LIN {X 0,Y 101.241,Z 307.493,A -85,B 0,C 180,E1 -26542.02,E2 -26542.02} C_VEL
LIN {X 0,Y 101.845,Z 307.419,A -85,B 0,C 180,E1 -26550,E2 -26550} C_VEL
LIN {X 0,Y 101.245,Z 307.494,A -85,B 0,C 180,E1 -26557.98,E2 -26557.98} C_VEL
LIN {X 0,Y 101.106,Z 307.516,A -85,B 0,C 180,E1 -26563.301,E2 -26563.301} C_VEL
LIN {X 0,Y 100.839,Z 307.548,A -85,B 0,C 180,E1 -26570.394,E2 -26570.394} C_VEL
LIN {X 0,Y 100.777,Z 307.552,A -85,B 0,C 180,E1 -26574.958,E2 -26574.958} C_VEL
LIN {X 0,Y 100.692,Z 307.562,A -85,B 0,C 180,E1 -26583.115,E2 -26583.115} C_VEL
LIN {X 0,Y 100.637,Z 307.573,A -85,B 0,C 180,E1 -26589.807,E2 -26589.807} C_VEL
LIN {X 0,Y 100.643,Z 307.573,A -85,B 0,C 180,E1 -26595.707,E2 -26595.707} C_VEL
LIN {X 0,Y 100.631,Z 307.568,A -85,B 0,C 180,E1 -26601.055,E2 -26601.055} C_VEL
LIN {X 0,Y 100.697,Z 307.564,A -85,B 0,C 180,E1 -26606.88,E2 -26606.88} C_VEL
LIN {X 0,Y 100.788,Z 307.552,A -85,B 0,C 180,E1 -26615.266,E2 -26615.266} C_VEL
LIN {X 0,Y 100.819,Z 307.55,A -85,B 0,C 180,E1 -26619.601,E2 -26619.601} C_VEL
LIN {X 0,Y 101.103,Z 307.511,A -85,B 0,C 180,E1 -26626.705,E2 -26626.705} C_VEL
LIN {X 0,Y 101.242,Z 307.495,A -85,B 0,C 180,E1 -26632.019,E2 -26632.019} C_VEL
LIN {X 0,Y 101.845,Z 307.421,A -85,B 0,C 180,E1 -26639.999,E2 -26639.999} C_VEL
LIN {X 0,Y 101.241,Z 307.496,A -85,B 0,C 180,E1 -26647.98,E2 -26647.98} C_VEL
LIN {X 0,Y 101.1,Z 307.516,A -85,B 0,C 180,E1 -26653.288,E2 -26653.288} C_VEL
LIN {X 0,Y 100.932,Z 307.538,A -85,B 0,C 180,E1 -26660.373,E2 -26660.373} C_VEL
LIN {X 0,Y 101.17,Z 307.509,A -85,B 0,C 180,E1 -26665.434,E2 -26665.434} C_VEL
LIN {X 0,Y 101.155,Z 307.514,A -85,B 0,C 180,E1 -26666.503,E2 -26666.503} C_VEL
LIN {X 0,Y 106.409,Z 325.53,A -85,B 0,C 180,E1 -26671.895,E2 -26671.895} C_VEL
LIN {X 0,Y 110.9,Z 342.326,A -85,B 0,C 180,E1 -26677.007,E2 -26677.007} C_VEL
LIN {X 0,Y 111.982,Z 348.423,A -85,B 0,C 180,E1 -26678.872,E2 -26678.872} C_VEL
LIN {X 0,Y 113.108,Z 364.062,A -85,B 0,C 180,E1 -26683.729,E2 -26683.729} C_VEL
LIN {X 0,Y 114.316,Z 378.581,A -85,B 0,C 180,E1 -26688.86,E2 -26688.86} C_VEL
LIN {X 0,Y 114.848,Z 387.278,A -85,B 0,C 180,E1 -26692.27,E2 -26692.27} C_VEL
LIN {X 0,Y 110.445,Z 398.562,A -85,B 0,C 180,E1 -26697.256,E2 -26697.256} C_VEL
LIN {X 0,Y 106.418,Z 409.833,A -85,B 0,C 180,E1 -26703.526,E2 -26703.526} C_VEL
LIN {X 0,Y 103.542,Z 419.322,A -85,B 0,C 180,E1 -26710.161,E2 -26710.161} C_VEL
LIN {X 0,Y 101.858,Z 427.24,A -85,B 0,C 180,E1 -26716.946,E2 -26716.946} C_VEL
LIN {X 0,Y 101.296,Z 433.952,A -85,B 0,C 180,E1 -26724.026,E2 -26724.026} C_VEL
LIN {X 0,Y 101.317,Z 438.583,A -85,B 0,C 180,E1 -26730,E2 -26730} C_VEL
LIN {X 0,Y 101.184,Z 440.994,A -85,B 0,C 180,E1 -26733.983,E2 -26733.983} C_VEL
LIN {X 0,Y 100.876,Z 444.648,A -85,B 0,C 180,E1 -26742.064,E2 -26742.064} C_VEL
LIN {X 0,Y 103.684,Z 448.473,A -85,B 0,C 180,E1 -26753.998,E2 -26753.998} C_VEL
LIN {X 0,Y 110.901,Z 450.872,A -85,B 0,C 180,E1 -26764.775,E2 -26764.775} C_VEL
LIN {X 0,Y 123.466,Z 452.199,A -85,B 0,C 180,E1 -26774.786,E2 -26774.786} C_VEL
LIN {X 0,Y 124.07,Z 452.003,A -85,B 0,C 180,E1 -26776.131,E2 -26776.131} C_VEL
LIN {X 0,Y 114.504,Z 448.317,A -85,B 0,C 180,E1 -26782.932,E2 -26782.932} C_VEL
LIN {X 0,Y 105.998,Z 442.642,A -85,B 0,C 180,E1 -26792.348,E2 -26792.348} C_VEL
LIN {X 0,Y 101.445,Z 436.258,A -85,B 0,C 180,E1 -26801.836,E2 -26801.836} C_VEL
LIN {X 0,Y 99.596,Z 428.977,A -85,B 0,C 180,E1 -26811.082,E2 -26811.082} C_VEL
LIN {X 0,Y 99.327,Z 422.478,A -85,B 0,C 180,E1 -26817.974,E2 -26817.974} C_VEL
LIN {X 0,Y 99.732,Z 414.622,A -85,B 0,C 180,E1 -26825.054,E2 -26825.054} C_VEL
LIN {X 0,Y 100.964,Z 405.332,A -85,B 0,C 180,E1 -26832.055,E2 -26832.055} C_VEL
LIN {X 0,Y 103.322,Z 394.429,A -85,B 0,C 180,E1 -26838.851,E2 -26838.851} C_VEL
LIN {X 0,Y 106.706,Z 381.556,A -85,B 0,C 180,E1 -26845.349,E2 -26845.349} C_VEL
LIN {X 0,Y 110.54,Z 368.745,A -85,B 0,C 180,E1 -26850.574,E2 -26850.574} C_VEL
LIN {X 0,Y 113.427,Z 359.141,A -85,B 0,C 180,E1 -26853.808,E2 -26853.808} C_VEL
LIN {X 0,Y 113.499,Z 356.487,A -85,B 0,C 180,E1 -26854.713,E2 -26854.713} C_VEL
LIN {X 0,Y 112.524,Z 353.993,A -85,B 0,C 180,E1 -26855.662,E2 -26855.662} C_VEL
LIN {X 0,Y 105.827,Z 345.177,A -85,B 0,C 180,E1 -26859.443,E2 -26859.443} C_VEL
LIN {X 0,Y 105.2,Z 343.541,A -85,B 0,C 180,E1 -26860.075,E2 -26860.075} C_VEL
LIN {X 0,Y 101.837,Z 331.883,A -85,B 0,C 180,E1 -26864.272,E2 -26864.272} C_VEL
LIN {X 0,Y 97.57,Z 319.143,A -85,B 0,C 180,E1 -26868.93,E2 -26868.93} C_VEL
LIN {X 0,Y 93.563,Z 308.455,A -85,B 0,C 180,E1 -26872.98,E2 -26872.98} C_VEL
LIN {X 0,Y 93.586,Z 308.453,A -85,B 0,C 180,E1 -26878.286,E2 -26878.286} C_VEL
LIN {X 0,Y 93.671,Z 308.44,A -85,B 0,C 180,E1 -26884.206,E2 -26884.206} C_VEL
LIN {X 0,Y 93.695,Z 308.434,A -85,B 0,C 180,E1 -26887.973,E2 -26887.973} C_VEL
LIN {X 0,Y 94.023,Z 308.394,A -85,B 0,C 180,E1 -26896.346,E2 -26896.346} C_VEL
LIN {X 0,Y 94.175,Z 308.376,A -85,B 0,C 180,E1 -26901.416,E2 -26901.416} C_VEL
LIN {X 0,Y 94.773,Z 308.299,A -85,B 0,C 180,E1 -26910,E2 -26910} C_VEL
LIN {X 0,Y 94.179,Z 308.373,A -85,B 0,C 180,E1 -26918.584,E2 -26918.584} C_VEL
LIN {X 0,Y 94.026,Z 308.399,A -85,B 0,C 180,E1 -26923.661,E2 -26923.661} C_VEL
LIN {X 0,Y 93.708,Z 308.437,A -85,B 0,C 180,E1 -26932.024,E2 -26932.024} C_VEL
LIN {X 0,Y 93.624,Z 308.441,A -85,B 0,C 180,E1 -26936.769,E2 -26936.769} C_VEL
LIN {X 0,Y 93.588,Z 308.444,A -85,B 0,C 180,E1 -26944.303,E2 -26944.303} C_VEL
LIN {X 0,Y 93.529,Z 308.452,A -85,B 0,C 180,E1 -26952.554,E2 -26952.554} C_VEL
LIN {X 0,Y 93.536,Z 308.456,A -85,B 0,C 180,E1 -26958.71,E2 -26958.71} C_VEL
LIN {X 0,Y 93.593,Z 308.451,A -85,B 0,C 180,E1 -26965.691,E2 -26965.691} C_VEL
LIN {X 0,Y 93.671,Z 308.442,A -85,B 0,C 180,E1 -26974.205,E2 -26974.205} C_VEL
LIN {X 0,Y 93.695,Z 308.432,A -85,B 0,C 180,E1 -26977.972,E2 -26977.972} C_VEL
LIN {X 0,Y 94.023,Z 308.392,A -85,B 0,C 180,E1 -26986.344,E2 -26986.344} C_VEL
LIN {X 0,Y 94.175,Z 308.378,A -85,B 0,C 180,E1 -26991.415,E2 -26991.415} C_VEL
LIN {X 0,Y 94.774,Z 308.301,A -85,B 0,C 180,E1 -26999.999,E2 -26999.999} C_VEL
LIN {X 0,Y 94.174,Z 308.375,A -85,B 0,C 180,E1 -27008.583,E2 -27008.583} C_VEL
LIN {X 0,Y 94.02,Z 308.398,A -85,B 0,C 180,E1 -27013.649,E2 -27013.649} C_VEL
LIN {X 0,Y 94.148,Z 308.467,A -85,B 0,C 180,E1 -27024.544,E2 -27024.544} C_VEL
LIN {X 0,Y 98.964,Z 324.412,A -85,B 0,C 180,E1 -27029.808,E2 -27029.808} C_VEL
LIN {X 0,Y 102.632,Z 338.427,A -85,B 0,C 180,E1 -27034.396,E2 -27034.396} C_VEL
LIN {X 0,Y 104.992,Z 348.076,A -85,B 0,C 180,E1 -27037.647,E2 -27037.647} C_VEL
LIN {X 0,Y 105.985,Z 363.218,A -85,B 0,C 180,E1 -27042.658,E2 -27042.658} C_VEL
LIN {X 0,Y 107.026,Z 376.793,A -85,B 0,C 180,E1 -27047.74,E2 -27047.74} C_VEL
LIN {X 0,Y 107.779,Z 386.56,A -85,B 0,C 180,E1 -27051.797,E2 -27051.797} C_VEL
LIN {X 0,Y 102.721,Z 399.394,A -85,B 0,C 180,E1 -27057.978,E2 -27057.978} C_VEL
LIN {X 0,Y 98.821,Z 410.31,A -85,B 0,C 180,E1 -27064.741,E2 -27064.741} C_VEL
LIN {X 0,Y 96.228,Z 419.271,A -85,B 0,C 180,E1 -27071.702,E2 -27071.702} C_VEL
LIN {X 0,Y 94.813,Z 427.268,A -85,B 0,C 180,E1 -27079.32,E2 -27079.32} C_VEL
LIN {X 0,Y 94.567,Z 432.8,A -85,B 0,C 180,E1 -27085.738,E2 -27085.738} C_VEL
LIN {X 0,Y 94.633,Z 435.92,A -85,B 0,C 180,E1 -27090,E2 -27090} C_VEL
LIN {X 0,Y 94.543,Z 438.515,A -85,B 0,C 180,E1 -27094.263,E2 -27094.263} C_VEL
LIN {X 0,Y 94.321,Z 442.289,A -85,B 0,C 180,E1 -27102.917,E2 -27102.917} C_VEL
LIN {X 0,Y 95.918,Z 445.194,A -85,B 0,C 180,E1 -27111.491,E2 -27111.491} C_VEL
LIN {X 0,Y 102.174,Z 448.295,A -85,B 0,C 180,E1 -27123.386,E2 -27123.386} C_VEL
LIN {X 0,Y 114.457,Z 450.423,A -85,B 0,C 180,E1 -27134.554,E2 -27134.554} C_VEL
LIN {X 0,Y 115.292,Z 450.49,A -85,B 0,C 180,E1 -27135.109,E2 -27135.109} C_VEL
LIN {X 0,Y 114.926,Z 450.16,A -85,B 0,C 180,E1 -27136.277,E2 -27136.277} C_VEL
LIN {X 0,Y 104.3,Z 444.98,A -85,B 0,C 180,E1 -27145.059,E2 -27145.059} C_VEL
LIN {X 0,Y 97.501,Z 439.096,A -85,B 0,C 180,E1 -27154.376,E2 -27154.376} C_VEL
LIN {X 0,Y 93.67,Z 431.835,A -85,B 0,C 180,E1 -27164.776,E2 -27164.776} C_VEL
LIN {X 0,Y 92.535,Z 424.247,A -85,B 0,C 180,E1 -27174.074,E2 -27174.074} C_VEL
LIN {X 0,Y 92.574,Z 416.247,A -85,B 0,C 180,E1 -27182.176,E2 -27182.176} C_VEL
LIN {X 0,Y 93.448,Z 407.303,A -85,B 0,C 180,E1 -27189.705,E2 -27189.705} C_VEL
LIN {X 0,Y 95.494,Z 396.741,A -85,B 0,C 180,E1 -27197.122,E2 -27197.122} C_VEL
LIN {X 0,Y 98.172,Z 386.288,A -85,B 0,C 180,E1 -27203.188,E2 -27203.188} C_VEL
LIN {X 0,Y 102.461,Z 371.979,A -85,B 0,C 180,E1 -27209.822,E2 -27209.822} C_VEL
LIN {X 0,Y 106.93,Z 357.501,A -85,B 0,C 180,E1 -27215.107,E2 -27215.107} C_VEL
LIN {X 0,Y 107.724,Z 354.824,A -85,B 0,C 180,E1 -27215.957,E2 -27215.957} C_VEL
LIN {X 0,Y 107.36,Z 351.95,A -85,B 0,C 180,E1 -27216.982,E2 -27216.982} C_VEL
LIN {X 0,Y 105.2,Z 343.541,A -85,B 0,C 180,E1 -27220.075,E2 -27220.075} C_VEL
LIN {X 0,Y 103.25,Z 339.032,A -85,B 0,C 180,E1 -27221.876,E2 -27221.876} C_VEL
LIN {X 0,Y 98.274,Z 332.395,A -85,B 0,C 180,E1 -27224.98,E2 -27224.98} C_VEL
LIN {X 0,Y 93.151,Z 325.723,A -85,B 0,C 180,E1 -27228.249,E2 -27228.249} C_VEL
LIN {X 0,Y 90.969,Z 321.134,A -85,B 0,C 180,E1 -27230.207,E2 -27230.207} C_VEL
LIN {X 0,Y 87.705,Z 312.585,A -85,B 0,C 180,E1 -27233.739,E2 -27233.739} C_VEL
LIN {X 0,Y 86.559,Z 309.328,A -85,B 0,C 180,E1 -27235.208,E2 -27235.208} C_VEL
LIN {X 0,Y 86.586,Z 309.324,A -85,B 0,C 180,E1 -27243.236,E2 -27243.236} C_VEL
LIN {X 0,Y 86.664,Z 309.315,A -85,B 0,C 180,E1 -27251.072,E2 -27251.072} C_VEL
LIN {X 0,Y 86.933,Z 309.275,A -85,B 0,C 180,E1 -27255.964,E2 -27255.964} C_VEL
LIN {X 0,Y 87.084,Z 309.26,A -85,B 0,C 180,E1 -27260.712,E2 -27260.712} C_VEL
LIN {X 0,Y 87.703,Z 309.18,A -85,B 0,C 180,E1 -27270,E2 -27270} C_VEL
LIN {X 0,Y 87.088,Z 309.255,A -85,B 0,C 180,E1 -27279.288,E2 -27279.288} C_VEL
LIN {X 0,Y 86.933,Z 309.281,A -85,B 0,C 180,E1 -27284.036,E2 -27284.036} C_VEL
LIN {X 0,Y 86.675,Z 309.308,A -85,B 0,C 180,E1 -27288.926,E2 -27288.926} C_VEL
LIN {X 0,Y 86.587,Z 309.318,A -85,B 0,C 180,E1 -27296.765,E2 -27296.765} C_VEL
LIN {X 0,Y 86.506,Z 309.329,A -85,B 0,C 180,E1 -27305.664,E2 -27305.664} C_VEL
LIN {X 0,Y 86.473,Z 309.331,A -85,B 0,C 180,E1 -27312.989,E2 -27312.989} C_VEL
LIN {X 0,Y 86.458,Z 309.335,A -85,B 0,C 180,E1 -27319.434,E2 -27319.434} C_VEL
LIN {X 0,Y 86.536,Z 309.33,A -85,B 0,C 180,E1 -27325.353,E2 -27325.353} C_VEL
LIN {X 0,Y 86.586,Z 309.324,A -85,B 0,C 180,E1 -27333.235,E2 -27333.235} C_VEL
LIN {X 0,Y 86.664,Z 309.315,A -85,B 0,C 180,E1 -27341.071,E2 -27341.071} C_VEL
LIN {X 0,Y 86.933,Z 309.274,A -85,B 0,C 180,E1 -27345.963,E2 -27345.963} C_VEL
LIN {X 0,Y 87.084,Z 309.261,A -85,B 0,C 180,E1 -27350.71,E2 -27350.71} C_VEL
LIN {X 0,Y 87.704,Z 309.182,A -85,B 0,C 180,E1 -27359.999,E2 -27359.999} C_VEL
LIN {X 0,Y 87.083,Z 309.256,A -85,B 0,C 180,E1 -27369.288,E2 -27369.288} C_VEL
LIN {X 0,Y 86.932,Z 309.282,A -85,B 0,C 180,E1 -27374.035,E2 -27374.035} C_VEL
LIN {X 0,Y 86.939,Z 309.487,A -85,B 0,C 180,E1 -27382.266,E2 -27382.266} C_VEL
LIN {X 0,Y 89.379,Z 315.622,A -85,B 0,C 180,E1 -27384.715,E2 -27384.715} C_VEL
LIN {X 0,Y 93.957,Z 332.136,A -85,B 0,C 180,E1 -27390.634,E2 -27390.634} C_VEL
LIN {X 0,Y 97.935,Z 348.364,A -85,B 0,C 180,E1 -27396.513,E2 -27396.513} C_VEL
LIN {X 0,Y 98.78,Z 359.544,A -85,B 0,C 180,E1 -27400.482,E2 -27400.482} C_VEL
LIN {X 0,Y 99.733,Z 374.228,A -85,B 0,C 180,E1 -27406.24,E2 -27406.24} C_VEL
LIN {X 0,Y 100.64,Z 385.256,A -85,B 0,C 180,E1 -27411.06,E2 -27411.06} C_VEL
LIN {X 0,Y 100.041,Z 387.443,A -85,B 0,C 180,E1 -27412.07,E2 -27412.07} C_VEL
LIN {X 0,Y 95.631,Z 398.35,A -85,B 0,C 180,E1 -27417.804,E2 -27417.804} C_VEL
LIN {X 0,Y 91.755,Z 409.225,A -85,B 0,C 180,E1 -27425.084,E2 -27425.084} C_VEL
LIN {X 0,Y 89.177,Z 418.376,A -85,B 0,C 180,E1 -27432.81,E2 -27432.81} C_VEL
LIN {X 0,Y 87.993,Z 426.095,A -85,B 0,C 180,E1 -27440.808,E2 -27440.808} C_VEL
LIN {X 0,Y 87.942,Z 431.553,A -85,B 0,C 180,E1 -27447.71,E2 -27447.71} C_VEL
LIN {X 0,Y 88.018,Z 434.577,A -85,B 0,C 180,E1 -27452.288,E2 -27452.288} C_VEL
LIN {X 0,Y 87.794,Z 436.965,A -85,B 0,C 180,E1 -27456.896,E2 -27456.896} C_VEL
LIN {X 0,Y 88.471,Z 441.434,A -85,B 0,C 180,E1 -27468.527,E2 -27468.527} C_VEL
LIN {X 0,Y 93.689,Z 445.264,A -85,B 0,C 180,E1 -27481.675,E2 -27481.675} C_VEL
LIN {X 0,Y 105.593,Z 448.176,A -85,B 0,C 180,E1 -27494.239,E2 -27494.239} C_VEL
LIN {X 0,Y 106.479,Z 448.292,A -85,B 0,C 180,E1 -27494.927,E2 -27494.927} C_VEL
LIN {X 0,Y 105.88,Z 447.81,A -85,B 0,C 180,E1 -27496.439,E2 -27496.439} C_VEL
LIN {X 0,Y 95.32,Z 441.675,A -85,B 0,C 180,E1 -27506.43,E2 -27506.43} C_VEL
LIN {X 0,Y 89.173,Z 434.988,A -85,B 0,C 180,E1 -27516.793,E2 -27516.793} C_VEL
LIN {X 0,Y 86.556,Z 428.573,A -85,B 0,C 180,E1 -27525.903,E2 -27525.903} C_VEL
LIN {X 0,Y 85.602,Z 420.959,A -85,B 0,C 180,E1 -27535.292,E2 -27535.292} C_VEL
LIN {X 0,Y 85.757,Z 412.911,A -85,B 0,C 180,E1 -27543.525,E2 -27543.525} C_VEL
LIN {X 0,Y 86.9,Z 403.42,A -85,B 0,C 180,E1 -27551.666,E2 -27551.666} C_VEL
LIN {X 0,Y 89.317,Z 392.485,A -85,B 0,C 180,E1 -27559.418,E2 -27559.418} C_VEL
LIN {X 0,Y 92.696,Z 380.196,A -85,B 0,C 180,E1 -27566.452,E2 -27566.452} C_VEL
LIN {X 0,Y 96.819,Z 367.226,A -85,B 0,C 180,E1 -27572.368,E2 -27572.368} C_VEL
LIN {X 0,Y 100.423,Z 355.958,A -85,B 0,C 180,E1 -27576.504,E2 -27576.504} C_VEL
LIN {X 0,Y 100.694,Z 354.457,A -85,B 0,C 180,E1 -27577.014,E2 -27577.014} C_VEL
LIN {X 0,Y 97.69,Z 342.679,A -85,B 0,C 180,E1 -27581.716,E2 -27581.716} C_VEL
LIN {X 0,Y 94.441,Z 331.581,A -85,B 0,C 180,E1 -27586.064,E2 -27586.064} C_VEL
LIN {X 0,Y 90.969,Z 321.134,A -85,B 0,C 180,E1 -27590.207,E2 -27590.207} C_VEL
LIN {X 0,Y 89.65,Z 318.266,A -85,B 0,C 180,E1 -27591.558,E2 -27591.558} C_VEL
LIN {X 0,Y 86.977,Z 314.923,A -85,B 0,C 180,E1 -27594.046,E2 -27594.046} C_VEL
LIN {X 0,Y 84.087,Z 312.601,A -85,B 0,C 180,E1 -27597.032,E2 -27597.032} C_VEL
LIN {X 0,Y 81.49,Z 311.111,A -85,B 0,C 180,E1 -27600.559,E2 -27600.559} C_VEL
LIN {X 0,Y 79.784,Z 310.346,A -85,B 0,C 180,E1 -27604.527,E2 -27604.527} C_VEL
LIN {X 0,Y 79.44,Z 310.203,A -85,B 0,C 180,E1 -27607.333,E2 -27607.333} C_VEL
LIN {X 0,Y 79.827,Z 310.159,A -85,B 0,C 180,E1 -27615.573,E2 -27615.573} C_VEL
LIN {X 0,Y 79.968,Z 310.149,A -85,B 0,C 180,E1 -27619.877,E2 -27619.877} C_VEL
LIN {X 0,Y 80.632,Z 310.06,A -85,B 0,C 180,E1 -27630,E2 -27630} C_VEL
LIN {X 0,Y 79.971,Z 310.141,A -85,B 0,C 180,E1 -27640.123,E2 -27640.123} C_VEL
LIN {X 0,Y 79.752,Z 310.174,A -85,B 0,C 180,E1 -27645.33,E2 -27645.33} C_VEL
LIN {X 0,Y 79.532,Z 310.202,A -85,B 0,C 180,E1 -27650.7,E2 -27650.7} C_VEL
LIN {X 0,Y 79.484,Z 310.205,A -85,B 0,C 180,E1 -27657.844,E2 -27657.844} C_VEL
LIN {X 0,Y 79.379,Z 310.22,A -85,B 0,C 180,E1 -27662.089,E2 -27662.089} C_VEL
LIN {X 0,Y 79.365,Z 310.224,A -85,B 0,C 180,E1 -27668.307,E2 -27668.307} C_VEL
LIN {X 0,Y 79.386,Z 310.22,A -85,B 0,C 180,E1 -27675.092,E2 -27675.092} C_VEL
LIN {X 0,Y 79.389,Z 310.218,A -85,B 0,C 180,E1 -27682.82,E2 -27682.82} C_VEL
LIN {X 0,Y 79.381,Z 310.216,A -85,B 0,C 180,E1 -27687.911,E2 -27687.911} C_VEL
LIN {X 0,Y 79.527,Z 310.204,A -85,B 0,C 180,E1 -27693.776,E2 -27693.776} C_VEL
LIN {X 0,Y 79.524,Z 310.202,A -85,B 0,C 180,E1 -27699.297,E2 -27699.297} C_VEL
LIN {X 0,Y 79.827,Z 310.158,A -85,B 0,C 180,E1 -27705.572,E2 -27705.572} C_VEL
LIN {X 0,Y 79.968,Z 310.149,A -85,B 0,C 180,E1 -27709.875,E2 -27709.875} C_VEL
LIN {X 0,Y 80.633,Z 310.062,A -85,B 0,C 180,E1 -27719.999,E2 -27719.999} C_VEL
LIN {X 0,Y 79.967,Z 310.141,A -85,B 0,C 180,E1 -27730.122,E2 -27730.122} C_VEL
LIN {X 0,Y 79.727,Z 310.172,A -85,B 0,C 180,E1 -27737.969,E2 -27737.969} C_VEL
LIN {X 0,Y 79.765,Z 310.321,A -85,B 0,C 180,E1 -27739.627,E2 -27739.627} C_VEL
LIN {X 0,Y 80.95,Z 313.289,A -85,B 0,C 180,E1 -27740.984,E2 -27740.984} C_VEL
LIN {X 0,Y 83.002,Z 317.673,A -85,B 0,C 180,E1 -27743.054,E2 -27743.054} C_VEL
LIN {X 0,Y 86.992,Z 332.784,A -85,B 0,C 180,E1 -27748.994,E2 -27748.994} C_VEL
LIN {X 0,Y 90.902,Z 349.065,A -85,B 0,C 180,E1 -27755.439,E2 -27755.439} C_VEL
LIN {X 0,Y 91.571,Z 355.389,A -85,B 0,C 180,E1 -27757.878,E2 -27757.878} C_VEL
LIN {X 0,Y 92.346,Z 370.194,A -85,B 0,C 180,E1 -27763.93,E2 -27763.93} C_VEL
LIN {X 0,Y 93.435,Z 383.884,A -85,B 0,C 180,E1 -27770.256,E2 -27770.256} C_VEL
LIN {X 0,Y 93.493,Z 385.333,A -85,B 0,C 180,E1 -27770.982,E2 -27770.982} C_VEL
LIN {X 0,Y 88.566,Z 397.166,A -85,B 0,C 180,E1 -27777.613,E2 -27777.613} C_VEL
LIN {X 0,Y 84.704,Z 408.022,A -85,B 0,C 180,E1 -27785.489,E2 -27785.489} C_VEL
LIN {X 0,Y 82.225,Z 417.145,A -85,B 0,C 180,E1 -27793.872,E2 -27793.872} C_VEL
LIN {X 0,Y 81.267,Z 424.781,A -85,B 0,C 180,E1 -27802.546,E2 -27802.546} C_VEL
LIN {X 0,Y 81.388,Z 430.184,A -85,B 0,C 180,E1 -27810,E2 -27810} C_VEL
LIN {X 0,Y 81.46,Z 433.054,A -85,B 0,C 180,E1 -27814.949,E2 -27814.949} C_VEL
LIN {X 0,Y 81.275,Z 435.277,A -85,B 0,C 180,E1 -27819.959,E2 -27819.959} C_VEL
LIN {X 0,Y 82.202,Z 438.889,A -85,B 0,C 180,E1 -27829.998,E2 -27829.998} C_VEL
LIN {X 0,Y 88.014,Z 442.921,A -85,B 0,C 180,E1 -27843.984,E2 -27843.984} C_VEL
LIN {X 0,Y 95.465,Z 445.118,A -85,B 0,C 180,E1 -27852.594,E2 -27852.594} C_VEL
LIN {X 0,Y 97.956,Z 445.445,A -85,B 0,C 180,E1 -27855.846,E2 -27855.846} C_VEL
LIN {X 0,Y 87.95,Z 439.083,A -85,B 0,C 180,E1 -27865.99,E2 -27865.99} C_VEL
LIN {X 0,Y 81.903,Z 431.86,A -85,B 0,C 180,E1 -27877.287,E2 -27877.287} C_VEL
LIN {X 0,Y 79.469,Z 425.01,A -85,B 0,C 180,E1 -27887.163,E2 -27887.163} C_VEL
LIN {X 0,Y 78.803,Z 418.911,A -85,B 0,C 180,E1 -27894.885,E2 -27894.885} C_VEL
LIN {X 0,Y 78.907,Z 410.622,A -85,B 0,C 180,E1 -27903.831,E2 -27903.831} C_VEL
LIN {X 0,Y 80.164,Z 400.841,A -85,B 0,C 180,E1 -27912.662,E2 -27912.662} C_VEL
LIN {X 0,Y 83.035,Z 388.724,A -85,B 0,C 180,E1 -27921.53,E2 -27921.53} C_VEL
LIN {X 0,Y 87.238,Z 374.657,A -85,B 0,C 180,E1 -27929.568,E2 -27929.568} C_VEL
LIN {X 0,Y 91.891,Z 360.802,A -85,B 0,C 180,E1 -27935.676,E2 -27935.676} C_VEL
LIN {X 0,Y 93.54,Z 355.698,A -85,B 0,C 180,E1 -27937.588,E2 -27937.588} C_VEL
LIN {X 0,Y 91.809,Z 347.96,A -85,B 0,C 180,E1 -27940.893,E2 -27940.893} C_VEL
LIN {X 0,Y 88.594,Z 336.323,A -85,B 0,C 180,E1 -27945.883,E2 -27945.883} C_VEL
LIN {X 0,Y 84.717,Z 324.168,A -85,B 0,C 180,E1 -27951.135,E2 -27951.135} C_VEL
LIN {X 0,Y 80.537,Z 313.186,A -85,B 0,C 180,E1 -27956.199,E2 -27956.199} C_VEL
LIN {X 0,Y 79.379,Z 310.222,A -85,B 0,C 180,E1 -27957.725,E2 -27957.725} C_VEL
LIN {X 0,Y 79.527,Z 310.203,A -85,B 0,C 180,E1 -27963.777,E2 -27963.777} C_VEL
LIN {X 0,Y 79.44,Z 310.203,A -85,B 0,C 180,E1 -27967.333,E2 -27967.333} C_VEL
LIN {X 0,Y 79.018,Z 310.267,A -85,B 0,C 180,E1 -27971.608,E2 -27971.608} C_VEL
LIN {X 0,Y 77.411,Z 310.474,A -85,B 0,C 180,E1 -27977.311,E2 -27977.311} C_VEL
LIN {X 0,Y 74.867,Z 310.789,A -85,B 0,C 180,E1 -27984.709,E2 -27984.709} C_VEL
LIN {X 0,Y 73.422,Z 310.953,A -85,B 0,C 180,E1 -27990.923,E2 -27990.923} C_VEL
LIN {X 0,Y 72.861,Z 311.03,A -85,B 0,C 180,E1 -28001.123,E2 -28001.123} C_VEL
LIN {X 0,Y 72.583,Z 311.062,A -85,B 0,C 180,E1 -28006.887,E2 -28006.887} C_VEL
LIN {X 0,Y 72.406,Z 311.091,A -85,B 0,C 180,E1 -28012.847,E2 -28012.847} C_VEL
LIN {X 0,Y 72.379,Z 311.093,A -85,B 0,C 180,E1 -28019.082,E2 -28019.082} C_VEL
LIN {X 0,Y 72.294,Z 311.099,A -85,B 0,C 180,E1 -28025.682,E2 -28025.682} C_VEL
LIN {X 0,Y 72.246,Z 311.103,A -85,B 0,C 180,E1 -28032.918,E2 -28032.918} C_VEL
LIN {X 0,Y 72.296,Z 311.097,A -85,B 0,C 180,E1 -28041.051,E2 -28041.051} C_VEL
LIN {X 0,Y 72.297,Z 311.104,A -85,B 0,C 180,E1 -28044.318,E2 -28044.318} C_VEL
LIN {X 0,Y 72.377,Z 311.091,A -85,B 0,C 180,E1 -28050.952,E2 -28050.952} C_VEL
LIN {X 0,Y 72.4,Z 311.083,A -85,B 0,C 180,E1 -28057.151,E2 -28057.151} C_VEL
LIN {X 0,Y 72.746,Z 311.04,A -85,B 0,C 180,E1 -28065.041,E2 -28065.041} C_VEL
LIN {X 0,Y 72.859,Z 311.034,A -85,B 0,C 180,E1 -28068.875,E2 -28068.875} C_VEL
LIN {X 0,Y 73.561,Z 310.943,A -85,B 0,C 180,E1 -28079.999,E2 -28079.999} C_VEL
LIN {X 0,Y 72.862,Z 311.027,A -85,B 0,C 180,E1 -28091.122,E2 -28091.122} C_VEL
LIN {X 0,Y 72.715,Z 311.2,A -85,B 0,C 180,E1 -28096.629,E2 -28096.629} C_VEL
LIN {X 0,Y 73.247,Z 313.064,A -85,B 0,C 180,E1 -28097.518,E2 -28097.518} C_VEL
LIN {X 0,Y 76.734,Z 320.348,A -85,B 0,C 180,E1 -28101.49,E2 -28101.49} C_VEL
LIN {X 0,Y 80.501,Z 335.226,A -85,B 0,C 180,E1 -28107.985,E2 -28107.985} C_VEL
LIN {X 0,Y 84.193,Z 351.181,A -85,B 0,C 180,E1 -28114.948,E2 -28114.948} C_VEL
LIN {X 0,Y 84.745,Z 359.47,A -85,B 0,C 180,E1 -28118.46,E2 -28118.46} C_VEL
LIN {X 0,Y 85.557,Z 373.998,A -85,B 0,C 180,E1 -28125.129,E2 -28125.129} C_VEL
LIN {X 0,Y 86.301,Z 383.803,A -85,B 0,C 180,E1 -28130.11,E2 -28130.11} C_VEL
LIN {X 0,Y 86.165,Z 385.06,A -85,B 0,C 180,E1 -28130.792,E2 -28130.792} C_VEL
LIN {X 0,Y 80.899,Z 397.519,A -85,B 0,C 180,E1 -28138.584,E2 -28138.584} C_VEL
LIN {X 0,Y 77.212,Z 408.242,A -85,B 0,C 180,E1 -28147.397,E2 -28147.397} C_VEL
LIN {X 0,Y 75.167,Z 416.962,A -85,B 0,C 180,E1 -28156.482,E2 -28156.482} C_VEL
LIN {X 0,Y 74.664,Z 423.367,A -85,B 0,C 180,E1 -28164.599,E2 -28164.599} C_VEL
LIN {X 0,Y 74.955,Z 428.66,A -85,B 0,C 180,E1 -28172.687,E2 -28172.687} C_VEL
LIN {X 0,Y 74.918,Z 431.289,A -85,B 0,C 180,E1 -28178.089,E2 -28178.089} C_VEL
LIN {X 0,Y 76.033,Z 436.181,A -85,B 0,C 180,E1 -28191.699,E2 -28191.699} C_VEL
LIN {X 0,Y 82.551,Z 440.439,A -85,B 0,C 180,E1 -28206.58,E2 -28206.58} C_VEL
LIN {X 0,Y 89.793,Z 442.634,A -85,B 0,C 180,E1 -28214.783,E2 -28214.783} C_VEL
LIN {X 0,Y 89.947,Z 442.599,A -85,B 0,C 180,E1 -28215.316,E2 -28215.316} C_VEL
LIN {X 0,Y 80.669,Z 436.18,A -85,B 0,C 180,E1 -28225.51,E2 -28225.51} C_VEL
LIN {X 0,Y 74.705,Z 428.412,A -85,B 0,C 180,E1 -28237.896,E2 -28237.896} C_VEL
LIN {X 0,Y 72.472,Z 420.985,A -85,B 0,C 180,E1 -28248.818,E2 -28248.818} C_VEL
LIN {X 0,Y 71.934,Z 414.418,A -85,B 0,C 180,E1 -28257.201,E2 -28257.201} C_VEL
LIN {X 0,Y 72.196,Z 406.81,A -85,B 0,C 180,E1 -28265.588,E2 -28265.588} C_VEL
LIN {X 0,Y 73.43,Z 397.951,A -85,B 0,C 180,E1 -28273.845,E2 -28273.845} C_VEL
LIN {X 0,Y 76.458,Z 386.257,A -85,B 0,C 180,E1 -28282.855,E2 -28282.855} C_VEL
LIN {X 0,Y 80.944,Z 371.996,A -85,B 0,C 180,E1 -28291.397,E2 -28291.397} C_VEL
LIN {X 0,Y 86.25,Z 356.701,A -85,B 0,C 180,E1 -28298.269,E2 -28298.269} C_VEL
LIN {X 0,Y 86.432,Z 355.464,A -85,B 0,C 180,E1 -28298.772,E2 -28298.772} C_VEL
LIN {X 0,Y 83.282,Z 343.211,A -85,B 0,C 180,E1 -28304.517,E2 -28304.517} C_VEL
LIN {X 0,Y 79.404,Z 330.081,A -85,B 0,C 180,E1 -28310.741,E2 -28310.741} C_VEL
LIN {X 0,Y 76.031,Z 320.383,A -85,B 0,C 180,E1 -28315.516,E2 -28315.516} C_VEL
LIN {X 0,Y 72.358,Z 311.095,A -85,B 0,C 180,E1 -28320.623,E2 -28320.623} C_VEL
LIN {X 0,Y 72.399,Z 311.084,A -85,B 0,C 180,E1 -28327.194,E2 -28327.194} C_VEL
LIN {X 0,Y 72.747,Z 311.04,A -85,B 0,C 180,E1 -28335.043,E2 -28335.043} C_VEL
LIN {X 0,Y 72.859,Z 311.034,A -85,B 0,C 180,E1 -28338.877,E2 -28338.877} C_VEL
LIN {X 0,Y 73.56,Z 310.941,A -85,B 0,C 180,E1 -28350,E2 -28350} C_VEL
LIN {X 0,Y 73.422,Z 310.953,A -85,B 0,C 180,E1 -28350.923,E2 -28350.923} C_VEL
LIN {X 0,Y 72.258,Z 311.11,A -85,B 0,C 180,E1 -28355.482,E2 -28355.482} C_VEL
LIN {X 0,Y 70.403,Z 311.34,A -85,B 0,C 180,E1 -28360.025,E2 -28360.025} C_VEL
LIN {X 0,Y 65.586,Z 311.939,A -85,B 0,C 180,E1 -28373.083,E2 -28373.083} C_VEL
LIN {X 0,Y 65.205,Z 311.976,A -85,B 0,C 180,E1 -28376.628,E2 -28376.628} C_VEL
LIN {X 0,Y 65.197,Z 311.983,A -85,B 0,C 180,E1 -28382.615,E2 -28382.615} C_VEL
LIN {X 0,Y 65.181,Z 311.985,A -85,B 0,C 180,E1 -28390.994,E2 -28390.994} C_VEL
LIN {X 0,Y 65.203,Z 311.981,A -85,B 0,C 180,E1 -28399.703,E2 -28399.703} C_VEL
LIN {X 0,Y 65.256,Z 311.974,A -85,B 0,C 180,E1 -28409.497,E2 -28409.497} C_VEL
LIN {X 0,Y 65.243,Z 311.981,A -85,B 0,C 180,E1 -28414.475,E2 -28414.475} C_VEL
LIN {X 0,Y 65.643,Z 311.926,A -85,B 0,C 180,E1 -28424.489,E2 -28424.489} C_VEL
LIN {X 0,Y 65.765,Z 311.915,A -85,B 0,C 180,E1 -28427.657,E2 -28427.657} C_VEL
LIN {X 0,Y 66.486,Z 311.824,A -85,B 0,C 180,E1 -28439.999,E2 -28439.999} C_VEL
LIN {X 0,Y 65.757,Z 311.918,A -85,B 0,C 180,E1 -28452.955,E2 -28452.955} C_VEL
LIN {X 0,Y 70.724,Z 323.771,A -85,B 0,C 180,E1 -28460.165,E2 -28460.165} C_VEL
LIN {X 0,Y 73.949,Z 337.485,A -85,B 0,C 180,E1 -28466.834,E2 -28466.834} C_VEL
LIN {X 0,Y 77.302,Z 352.617,A -85,B 0,C 180,E1 -28474.146,E2 -28474.146} C_VEL
LIN {X 0,Y 77.763,Z 359.383,A -85,B 0,C 180,E1 -28477.306,E2 -28477.306} C_VEL
LIN {X 0,Y 78.439,Z 374.063,A -85,B 0,C 180,E1 -28484.662,E2 -28484.662} C_VEL
LIN {X 0,Y 79.174,Z 383.562,A -85,B 0,C 180,E1 -28489.942,E2 -28489.942} C_VEL
LIN {X 0,Y 74.348,Z 395.039,A -85,B 0,C 180,E1 -28497.633,E2 -28497.633} C_VEL
LIN {X 0,Y 70.684,Z 405.279,A -85,B 0,C 180,E1 -28506.564,E2 -28506.564} C_VEL
LIN {X 0,Y 68.559,Z 414.333,A -85,B 0,C 180,E1 -28516.664,E2 -28516.664} C_VEL
LIN {X 0,Y 68.158,Z 421.835,A -85,B 0,C 180,E1 -28527.044,E2 -28527.044} C_VEL
LIN {X 0,Y 68.501,Z 425.43,A -85,B 0,C 180,E1 -28532.94,E2 -28532.94} C_VEL
LIN {X 0,Y 68.635,Z 426.946,A -85,B 0,C 180,E1 -28535.877,E2 -28535.877} C_VEL
LIN {X 0,Y 68.608,Z 429.395,A -85,B 0,C 180,E1 -28541.822,E2 -28541.822} C_VEL
LIN {X 0,Y 71.803,Z 434.968,A -85,B 0,C 180,E1 -28559.301,E2 -28559.301} C_VEL
LIN {X 0,Y 81.018,Z 439.011,A -85,B 0,C 180,E1 -28573.945,E2 -28573.945} C_VEL
LIN {X 0,Y 80.798,Z 438.582,A -85,B 0,C 180,E1 -28575.906,E2 -28575.906} C_VEL
LIN {X 0,Y 71.996,Z 431.412,A -85,B 0,C 180,E1 -28587.529,E2 -28587.529} C_VEL
LIN {X 0,Y 66.878,Z 422.787,A -85,B 0,C 180,E1 -28601.625,E2 -28601.625} C_VEL
LIN {X 0,Y 65.439,Z 415.509,A -85,B 0,C 180,E1 -28612.286,E2 -28612.286} C_VEL
LIN {X 0,Y 65.172,Z 408.199,A -85,B 0,C 180,E1 -28621.546,E2 -28621.546} C_VEL
LIN {X 0,Y 66.244,Z 398.131,A -85,B 0,C 180,E1 -28632.252,E2 -28632.252} C_VEL
LIN {X 0,Y 69.349,Z 385.566,A -85,B 0,C 180,E1 -28643.016,E2 -28643.016} C_VEL
LIN {X 0,Y 73.572,Z 372.399,A -85,B 0,C 180,E1 -28651.696,E2 -28651.696} C_VEL
LIN {X 0,Y 78.653,Z 358.351,A -85,B 0,C 180,E1 -28658.719,E2 -28658.719} C_VEL
LIN {X 0,Y 79.343,Z 356.275,A -85,B 0,C 180,E1 -28659.581,E2 -28659.581} C_VEL
LIN {X 0,Y 76.098,Z 343.515,A -85,B 0,C 180,E1 -28666.159,E2 -28666.159} C_VEL
LIN {X 0,Y 72.547,Z 331.358,A -85,B 0,C 180,E1 -28672.562,E2 -28672.562} C_VEL
LIN {X 0,Y 69.3,Z 321.883,A -85,B 0,C 180,E1 -28677.831,E2 -28677.831} C_VEL
LIN {X 0,Y 66.086,Z 314.474,A -85,B 0,C 180,E1 -28682.551,E2 -28682.551} C_VEL
LIN {X 0,Y 65.256,Z 311.979,A -85,B 0,C 180,E1 -28684.196,E2 -28684.196} C_VEL
LIN {X 0,Y 65.644,Z 311.925,A -85,B 0,C 180,E1 -28694.491,E2 -28694.491} C_VEL
LIN {X 0,Y 65.765,Z 311.917,A -85,B 0,C 180,E1 -28697.659,E2 -28697.659} C_VEL
LIN {X 0,Y 66.485,Z 311.822,A -85,B 0,C 180,E1 -28710,E2 -28710} C_VEL
LIN {X 0,Y 65.766,Z 311.917,A -85,B 0,C 180,E1 -28722.341,E2 -28722.341} C_VEL
LIN {X 0,Y 65.39,Z 311.958,A -85,B 0,C 180,E1 -28728.811,E2 -28728.811} C_VEL
LIN {X 0,Y 65.205,Z 311.976,A -85,B 0,C 180,E1 -28736.628,E2 -28736.628} C_VEL
LIN {X 0,Y 64.801,Z 312.038,A -85,B 0,C 180,E1 -28740.071,E2 -28740.071} C_VEL
LIN {X 0,Y 63.354,Z 312.214,A -85,B 0,C 180,E1 -28745.207,E2 -28745.207} C_VEL
LIN {X 0,Y 60.107,Z 312.621,A -85,B 0,C 180,E1 -28754.077,E2 -28754.077} C_VEL
LIN {X 0,Y 58.247,Z 312.847,A -85,B 0,C 180,E1 -28761.84,E2 -28761.84} C_VEL
LIN {X 0,Y 58.059,Z 312.865,A -85,B 0,C 180,E1 -28765.883,E2 -28765.883} C_VEL
LIN {X 0,Y 58.153,Z 312.862,A -85,B 0,C 180,E1 -28771.09,E2 -28771.09} C_VEL
LIN {X 0,Y 58.531,Z 312.813,A -85,B 0,C 180,E1 -28783.861,E2 -28783.861} C_VEL
LIN {X 0,Y 58.8,Z 312.777,A -85,B 0,C 180,E1 -28793.134,E2 -28793.134} C_VEL
LIN {X 0,Y 59.377,Z 312.71,A -85,B 0,C 180,E1 -28799.998,E2 -28799.998} C_VEL
LIN {X 0,Y 58.763,Z 312.987,A -85,B 0,C 180,E1 -28808.813,E2 -28808.813} C_VEL
LIN {X 0,Y 59.408,Z 315.105,A -85,B 0,C 180,E1 -28810.22,E2 -28810.22} C_VEL
LIN {X 0,Y 61.283,Z 319.049,A -85,B 0,C 180,E1 -28813.258,E2 -28813.258} C_VEL
LIN {X 0,Y 64.763,Z 327.663,A -85,B 0,C 180,E1 -28818.998,E2 -28818.998} C_VEL
LIN {X 0,Y 67.959,Z 342.185,A -85,B 0,C 180,E1 -28826.899,E2 -28826.899} C_VEL
LIN {X 0,Y 70.695,Z 355.941,A -85,B 0,C 180,E1 -28834.302,E2 -28834.302} C_VEL
LIN {X 0,Y 71.114,Z 370.113,A -85,B 0,C 180,E1 -28841.895,E2 -28841.895} C_VEL
LIN {X 0,Y 71.949,Z 383.019,A -85,B 0,C 180,E1 -28849.674,E2 -28849.674} C_VEL
LIN {X 0,Y 67.405,Z 393.509,A -85,B 0,C 180,E1 -28857.429,E2 -28857.429} C_VEL
LIN {X 0,Y 63.751,Z 403.699,A -85,B 0,C 180,E1 -28867.303,E2 -28867.303} C_VEL
LIN {X 0,Y 61.826,Z 412.72,A -85,B 0,C 180,E1 -28878.525,E2 -28878.525} C_VEL
LIN {X 0,Y 61.824,Z 420.208,A -85,B 0,C 180,E1 -28890,E2 -28890} C_VEL
LIN {X 0,Y 62.295,Z 423.674,A -85,B 0,C 180,E1 -28896.478,E2 -28896.478} C_VEL
LIN {X 0,Y 62.396,Z 426.21,A -85,B 0,C 180,E1 -28903.019,E2 -28903.019} C_VEL
LIN {X 0,Y 66.237,Z 431.96,A -85,B 0,C 180,E1 -28922.041,E2 -28922.041} C_VEL
LIN {X 0,Y 72.419,Z 434.95,A -85,B 0,C 180,E1 -28932.791,E2 -28932.791} C_VEL
LIN {X 0,Y 72.915,Z 434.83,A -85,B 0,C 180,E1 -28935.431,E2 -28935.431} C_VEL
LIN {X 0,Y 63.547,Z 426.041,A -85,B 0,C 180,E1 -28950.155,E2 -28950.155} C_VEL
LIN {X 0,Y 59.614,Z 417.597,A -85,B 0,C 180,E1 -28964.374,E2 -28964.374} C_VEL
LIN {X 0,Y 58.652,Z 411.834,A -85,B 0,C 180,E1 -28973.12,E2 -28973.12} C_VEL
LIN {X 0,Y 58.459,Z 404.041,A -85,B 0,C 180,E1 -28983.448,E2 -28983.448} C_VEL
LIN {X 0,Y 59.594,Z 394.989,A -85,B 0,C 180,E1 -28993.644,E2 -28993.644} C_VEL
LIN {X 0,Y 62.843,Z 382.894,A -85,B 0,C 180,E1 -29004.691,E2 -29004.691} C_VEL
LIN {X 0,Y 67.895,Z 368.257,A -85,B 0,C 180,E1 -29014.705,E2 -29014.705} C_VEL
LIN {X 0,Y 72.103,Z 356.98,A -85,B 0,C 180,E1 -29020.535,E2 -29020.535} C_VEL
LIN {X 0,Y 69.678,Z 346.729,A -85,B 0,C 180,E1 -29026.384,E2 -29026.384} C_VEL
LIN {X 0,Y 66.337,Z 334.623,A -85,B 0,C 180,E1 -29033.421,E2 -29033.421} C_VEL
LIN {X 0,Y 63.02,Z 324.409,A -85,B 0,C 180,E1 -29039.865,E2 -29039.865} C_VEL
LIN {X 0,Y 59.676,Z 316.433,A -85,B 0,C 180,E1 -29045.657,E2 -29045.657} C_VEL
LIN {X 0,Y 58.354,Z 313.744,A -85,B 0,C 180,E1 -29047.891,E2 -29047.891} C_VEL
LIN {X 0,Y 58.193,Z 312.858,A -85,B 0,C 180,E1 -29048.758,E2 -29048.758} C_VEL
LIN {X 0,Y 58.647,Z 312.798,A -85,B 0,C 180,E1 -29056.133,E2 -29056.133} C_VEL
LIN {X 0,Y 58.799,Z 312.777,A -85,B 0,C 180,E1 -29063.135,E2 -29063.135} C_VEL
LIN {X 0,Y 59.376,Z 312.707,A -85,B 0,C 180,E1 -29070,E2 -29070} C_VEL
LIN {X 0,Y 58.803,Z 312.783,A -85,B 0,C 180,E1 -29076.865,E2 -29076.865} C_VEL
LIN {X 0,Y 58.533,Z 312.813,A -85,B 0,C 180,E1 -29086.14,E2 -29086.14} C_VEL
LIN {X 0,Y 58.154,Z 312.865,A -85,B 0,C 180,E1 -29098.909,E2 -29098.909} C_VEL
LIN {X 0,Y 58.159,Z 312.861,A -85,B 0,C 180,E1 -29102.229,E2 -29102.229} C_VEL
LIN {X 0,Y 58.031,Z 312.88,A -85,B 0,C 180,E1 -29107.268,E2 -29107.268} C_VEL
LIN {X 0,Y 58.012,Z 312.884,A -85,B 0,C 180,E1 -29116.627,E2 -29116.627} C_VEL
LIN {X 0,Y 58.059,Z 312.865,A -85,B 0,C 180,E1 -29125.883,E2 -29125.883} C_VEL
LIN {X 0,Y 57.832,Z 312.899,A -85,B 0,C 180,E1 -29129.739,E2 -29129.739} C_VEL
LIN {X 0,Y 57.058,Z 313.003,A -85,B 0,C 180,E1 -29133.575,E2 -29133.575} C_VEL
LIN {X 0,Y 55.342,Z 313.22,A -85,B 0,C 180,E1 -29139.407,E2 -29139.407} C_VEL
LIN {X 0,Y 51.981,Z 313.627,A -85,B 0,C 180,E1 -29154.431,E2 -29154.431} C_VEL
LIN {X 0,Y 52.129,Z 313.604,A -85,B 0,C 180,E1 -29158.976,E2 -29158.976} C_VEL
LIN {X 0,Y 51.96,Z 313.63,A -85,B 0,C 180,E1 -29162.906,E2 -29162.906} C_VEL
LIN {X 0,Y 52.058,Z 314.513,A -85,B 0,C 180,E1 -29163.869,E2 -29163.869} C_VEL
LIN {X 0,Y 55.864,Z 323.463,A -85,B 0,C 180,E1 -29171.795,E2 -29171.795} C_VEL
LIN {X 0,Y 58.648,Z 330.989,A -85,B 0,C 180,E1 -29177.431,E2 -29177.431} C_VEL
LIN {X 0,Y 61.28,Z 344.036,A -85,B 0,C 180,E1 -29185.47,E2 -29185.47} C_VEL
LIN {X 0,Y 63.796,Z 357.136,A -85,B 0,C 180,E1 -29193.421,E2 -29193.421} C_VEL
LIN {X 0,Y 64.102,Z 371.662,A -85,B 0,C 180,E1 -29202.183,E2 -29202.183} C_VEL
LIN {X 0,Y 64.726,Z 382.298,A -85,B 0,C 180,E1 -29209.346,E2 -29209.346} C_VEL
LIN {X 0,Y 59.446,Z 394.523,A -85,B 0,C 180,E1 -29219.837,E2 -29219.837} C_VEL
LIN {X 0,Y 56.157,Z 404.768,A -85,B 0,C 180,E1 -29231.767,E2 -29231.767} C_VEL
LIN {X 0,Y 55.174,Z 413.327,A -85,B 0,C 180,E1 -29244.518,E2 -29244.518} C_VEL
LIN {X 0,Y 55.69,Z 418.43,A -85,B 0,C 180,E1 -29253.618,E2 -29253.618} C_VEL
LIN {X 0,Y 56.026,Z 420.171,A -85,B 0,C 180,E1 -29257.206,E2 -29257.206} C_VEL
LIN {X 0,Y 56.22,Z 421.629,A -85,B 0,C 180,E1 -29260.808,E2 -29260.808} C_VEL
LIN {X 0,Y 58.518,Z 427.036,A -85,B 0,C 180,E1 -29278.711,E2 -29278.711} C_VEL
LIN {X 0,Y 65.021,Z 430.883,A -85,B 0,C 180,E1 -29292.738,E2 -29292.738} C_VEL
LIN {X 0,Y 64.521,Z 430.225,A -85,B 0,C 180,E1 -29295.583,E2 -29295.583} C_VEL
LIN {X 0,Y 56.453,Z 421.921,A -85,B 0,C 180,E1 -29310.136,E2 -29310.136} C_VEL
LIN {X 0,Y 53.187,Z 414.927,A -85,B 0,C 180,E1 -29322.706,E2 -29322.706} C_VEL
LIN {X 0,Y 51.905,Z 407.854,A -85,B 0,C 180,E1 -29334.173,E2 -29334.173} C_VEL
LIN {X 0,Y 52.011,Z 398.059,A -85,B 0,C 180,E1 -29347.768,E2 -29347.768} C_VEL
LIN {X 0,Y 54.401,Z 386.468,A -85,B 0,C 180,E1 -29360.812,E2 -29360.812} C_VEL
LIN {X 0,Y 57.998,Z 375.19,A -85,B 0,C 180,E1 -29370.64,E2 -29370.64} C_VEL
LIN {X 0,Y 62.861,Z 362.595,A -85,B 0,C 180,E1 -29378.967,E2 -29378.967} C_VEL
LIN {X 0,Y 64.732,Z 357.839,A -85,B 0,C 180,E1 -29381.531,E2 -29381.531} C_VEL
LIN {X 0,Y 64.872,Z 356.655,A -85,B 0,C 180,E1 -29382.187,E2 -29382.187} C_VEL
LIN {X 0,Y 62.112,Z 345.473,A -85,B 0,C 180,E1 -29389.412,E2 -29389.412} C_VEL
LIN {X 0,Y 58.97,Z 333.779,A -85,B 0,C 180,E1 -29397.162,E2 -29397.162} C_VEL
LIN {X 0,Y 55.904,Z 324.845,A -85,B 0,C 180,E1 -29403.896,E2 -29403.896} C_VEL
LIN {X 0,Y 54.332,Z 320.911,A -85,B 0,C 180,E1 -29407.166,E2 -29407.166} C_VEL
LIN {X 0,Y 51.579,Z 314.669,A -85,B 0,C 180,E1 -29413.159,E2 -29413.159} C_VEL
LIN {X 0,Y 51.467,Z 313.691,A -85,B 0,C 180,E1 -29414.151,E2 -29414.151} C_VEL
LIN {X 0,Y 51.679,Z 313.664,A -85,B 0,C 180,E1 -29422.184,E2 -29422.184} C_VEL
LIN {X 0,Y 52.26,Z 313.593,A -85,B 0,C 180,E1 -29430,E2 -29430} C_VEL
LIN {X 0,Y 51.682,Z 313.666,A -85,B 0,C 180,E1 -29437.816,E2 -29437.816} C_VEL
LIN {X 0,Y 51.4,Z 313.699,A -85,B 0,C 180,E1 -29446.832,E2 -29446.832} C_VEL
LIN {X 0,Y 51.028,Z 313.747,A -85,B 0,C 180,E1 -29454.406,E2 -29454.406} C_VEL
LIN {X 0,Y 51.005,Z 313.747,A -85,B 0,C 180,E1 -29464.231,E2 -29464.231} C_VEL
LIN {X 0,Y 50.979,Z 313.76,A -85,B 0,C 180,E1 -29476.422,E2 -29476.422} C_VEL
LIN {X 0,Y 51.051,Z 313.747,A -85,B 0,C 180,E1 -29486.585,E2 -29486.585} C_VEL
LIN {X 0,Y 51.027,Z 313.747,A -85,B 0,C 180,E1 -29495.592,E2 -29495.592} C_VEL
LIN {X 0,Y 51.473,Z 313.691,A -85,B 0,C 180,E1 -29504.151,E2 -29504.151} C_VEL
LIN {X 0,Y 51.679,Z 313.666,A -85,B 0,C 180,E1 -29512.182,E2 -29512.182} C_VEL
LIN {X 0,Y 52.129,Z 313.604,A -85,B 0,C 180,E1 -29518.976,E2 -29518.976} C_VEL
LIN {X 0,Y 52.709,Z 314.316,A -85,B 0,C 180,E1 -29522.395,E2 -29522.395} C_VEL
LIN {X 0,Y 53.628,Z 316.721,A -85,B 0,C 180,E1 -29526.061,E2 -29526.061} C_VEL
LIN {X 0,Y 54.457,Z 320.578,A -85,B 0,C 180,E1 -29529.255,E2 -29529.255} C_VEL
LIN {X 0,Y 54.534,Z 325.245,A -85,B 0,C 180,E1 -29531.788,E2 -29531.788} C_VEL
LIN {X 0,Y 53.317,Z 337.505,A -85,B 0,C 180,E1 -29538.011,E2 -29538.011} C_VEL
LIN {X 0,Y 53.488,Z 339.416,A -85,B 0,C 180,E1 -29539.298,E2 -29539.298} C_VEL
LIN {X 0,Y 55.584,Z 351.51,A -85,B 0,C 180,E1 -29547.737,E2 -29547.737} C_VEL
LIN {X 0,Y 56.862,Z 358.778,A -85,B 0,C 180,E1 -29552.732,E2 -29552.732} C_VEL
LIN {X 0,Y 57.056,Z 372.732,A -85,B 0,C 180,E1 -29562.347,E2 -29562.347} C_VEL
LIN {X 0,Y 57.63,Z 380.988,A -85,B 0,C 180,E1 -29568.592,E2 -29568.592} C_VEL
LIN {X 0,Y 52.565,Z 392.757,A -85,B 0,C 180,E1 -29579.908,E2 -29579.908} C_VEL
LIN {X 0,Y 49.405,Z 402.965,A -85,B 0,C 180,E1 -29593.47,E2 -29593.47} C_VEL
LIN {X 0,Y 48.902,Z 411.485,A -85,B 0,C 180,E1 -29607.941,E2 -29607.941} C_VEL
LIN {X 0,Y 49.809,Z 416.47,A -85,B 0,C 180,E1 -29618.111,E2 -29618.111} C_VEL
LIN {X 0,Y 50.034,Z 417.475,A -85,B 0,C 180,E1 -29620.51,E2 -29620.51} C_VEL
LIN {X 0,Y 50.684,Z 420.495,A -85,B 0,C 180,E1 -29630.283,E2 -29630.283} C_VEL
LIN {X 0,Y 55.885,Z 425.526,A -85,B 0,C 180,E1 -29648.961,E2 -29648.961} C_VEL
LIN {X 0,Y 58.072,Z 426.58,A -85,B 0,C 180,E1 -29653.439,E2 -29653.439} C_VEL
LIN {X 0,Y 49.364,Z 417.302,A -85,B 0,C 180,E1 -29670.507,E2 -29670.507} C_VEL
LIN {X 0,Y 46.264,Z 409.931,A -85,B 0,C 180,E1 -29684.585,E2 -29684.585} C_VEL
LIN {X 0,Y 45.053,Z 402.132,A -85,B 0,C 180,E1 -29697.767,E2 -29697.767} C_VEL
LIN {X 0,Y 45.583,Z 393.083,A -85,B 0,C 180,E1 -29711.114,E2 -29711.114} C_VEL
LIN {X 0,Y 48.776,Z 380.778,A -85,B 0,C 180,E1 -29725.614,E2 -29725.614} C_VEL
LIN {X 0,Y 54.306,Z 366.122,A -85,B 0,C 180,E1 -29737.983,E2 -29737.983} C_VEL
LIN {X 0,Y 57.564,Z 358.109,A -85,B 0,C 180,E1 -29742.988,E2 -29742.988} C_VEL
LIN {X 0,Y 57.243,Z 355.051,A -85,B 0,C 180,E1 -29745.096,E2 -29745.096} C_VEL
LIN {X 0,Y 54.347,Z 343.025,A -85,B 0,C 180,E1 -29753.957,E2 -29753.957} C_VEL
LIN {X 0,Y 51.723,Z 333.332,A -85,B 0,C 180,E1 -29761.604,E2 -29761.604} C_VEL
LIN {X 0,Y 48.962,Z 325.322,A -85,B 0,C 180,E1 -29768.956,E2 -29768.956} C_VEL
LIN {X 0,Y 46.058,Z 318.311,A -85,B 0,C 180,E1 -29776.769,E2 -29776.769} C_VEL
LIN {X 0,Y 45.194,Z 317.012,A -85,B 0,C 180,E1 -29778.791,E2 -29778.791} C_VEL
LIN {X 0,Y 44.569,Z 314.55,A -85,B 0,C 180,E1 -29781.784,E2 -29781.784} C_VEL
LIN {X 0,Y 45.136,Z 314.48,A -85,B 0,C 180,E1 -29790,E2 -29790} C_VEL
LIN {X 0,Y 44.538,Z 314.553,A -85,B 0,C 180,E1 -29799.08,E2 -29799.08} C_VEL
LIN {X 0,Y 44.176,Z 314.599,A -85,B 0,C 180,E1 -29808.554,E2 -29808.554} C_VEL
LIN {X 0,Y 43.845,Z 314.645,A -85,B 0,C 180,E1 -29818.743,E2 -29818.743} C_VEL
LIN {X 0,Y 43.793,Z 314.651,A -85,B 0,C 180,E1 -29829.937,E2 -29829.937} C_VEL
LIN {X 0,Y 43.842,Z 314.645,A -85,B 0,C 180,E1 -29843.276,E2 -29843.276} C_VEL
LIN {X 0,Y 43.845,Z 314.644,A -85,B 0,C 180,E1 -29851.254,E2 -29851.254} C_VEL
LIN {X 0,Y 44.257,Z 314.596,A -85,B 0,C 180,E1 -29862.33,E2 -29862.33} C_VEL
LIN {X 0,Y 44.738,Z 314.529,A -85,B 0,C 180,E1 -29874.928,E2 -29874.928} C_VEL
LIN {X 0,Y 44.779,Z 314.665,A -85,B 0,C 180,E1 -29875.497,E2 -29875.497} C_VEL
LIN {X 0,Y 45.507,Z 316.543,A -85,B 0,C 180,E1 -29877.785,E2 -29877.785} C_VEL
LIN {X 0,Y 46.517,Z 317.865,A -85,B 0,C 180,E1 -29879.998,E2 -29879.998} C_VEL
LIN {X 0,Y 49.735,Z 325.882,A -85,B 0,C 180,E1 -29888.442,E2 -29888.442} C_VEL
LIN {X 0,Y 52.505,Z 334.048,A -85,B 0,C 180,E1 -29895.526,E2 -29895.526} C_VEL
LIN {X 0,Y 53.488,Z 339.416,A -85,B 0,C 180,E1 -29899.298,E2 -29899.298} C_VEL
LIN {X 0,Y 53.688,Z 344.562,A -85,B 0,C 180,E1 -29902.591,E2 -29902.591} C_VEL
LIN {X 0,Y 53.016,Z 349.778,A -85,B 0,C 180,E1 -29905.635,E2 -29905.635} C_VEL
LIN {X 0,Y 50.694,Z 360.09,A -85,B 0,C 180,E1 -29911.991,E2 -29911.991} C_VEL
LIN {X 0,Y 49.858,Z 366.788,A -85,B 0,C 180,E1 -29916.967,E2 -29916.967} C_VEL
LIN {X 0,Y 50.376,Z 380.433,A -85,B 0,C 180,E1 -29928.495,E2 -29928.495} C_VEL
LIN {X 0,Y 45.129,Z 392.41,A -85,B 0,C 180,E1 -29942.147,E2 -29942.147} C_VEL
LIN {X 0,Y 42.566,Z 402.347,A -85,B 0,C 180,E1 -29958.089,E2 -29958.089} C_VEL
LIN {X 0,Y 43.013,Z 410.181,A -85,B 0,C 180,E1 -29973.742,E2 -29973.742} C_VEL
LIN {X 0,Y 44.022,Z 413.7,A -85,B 0,C 180,E1 -29981.965,E2 -29981.965} C_VEL
LIN {X 0,Y 44.613,Z 415.867,A -85,B 0,C 180,E1 -29989.061,E2 -29989.061} C_VEL
LIN {X 0,Y 50.495,Z 421.679,A -85,B 0,C 180,E1 -30011.879,E2 -30011.879} C_VEL
LIN {X 0,Y 49.273,Z 420.561,A -85,B 0,C 180,E1 -30014.509,E2 -30014.509} C_VEL
LIN {X 0,Y 41.927,Z 411.566,A -85,B 0,C 180,E1 -30032.553,E2 -30032.553} C_VEL
LIN {X 0,Y 39.266,Z 404.418,A -85,B 0,C 180,E1 -30047.074,E2 -30047.074} C_VEL
LIN {X 0,Y 38.493,Z 394.329,A -85,B 0,C 180,E1 -30065.24,E2 -30065.24} C_VEL
LIN {X 0,Y 40.868,Z 382.367,A -85,B 0,C 180,E1 -30082.766,E2 -30082.766} C_VEL
LIN {X 0,Y 45.651,Z 369.256,A -85,B 0,C 180,E1 -30096.626,E2 -30096.626} C_VEL
LIN {X 0,Y 50.189,Z 358.83,A -85,B 0,C 180,E1 -30104.442,E2 -30104.442} C_VEL
LIN {X 0,Y 50.286,Z 356.219,A -85,B 0,C 180,E1 -30106.397,E2 -30106.397} C_VEL
LIN {X 0,Y 47.613,Z 344.498,A -85,B 0,C 180,E1 -30116.391,E2 -30116.391} C_VEL
LIN {X 0,Y 45.598,Z 336.274,A -85,B 0,C 180,E1 -30123.928,E2 -30123.928} C_VEL
LIN {X 0,Y 43.466,Z 329.523,A -85,B 0,C 180,E1 -30131.133,E2 -30131.133} C_VEL
LIN {X 0,Y 40.897,Z 322.65,A -85,B 0,C 180,E1 -30140.105,E2 -30140.105} C_VEL
LIN {X 0,Y 39.732,Z 319.566,A -85,B 0,C 180,E1 -30144.926,E2 -30144.926} C_VEL
LIN {X 0,Y 37.688,Z 315.41,A -85,B 0,C 180,E1 -30153.676,E2 -30153.676} C_VEL
LIN {X 0,Y 37.335,Z 315.451,A -85,B 0,C 180,E1 -30160.851,E2 -30160.851} C_VEL
LIN {X 0,Y 37.07,Z 315.483,A -85,B 0,C 180,E1 -30168.56,E2 -30168.56} C_VEL
LIN {X 0,Y 36.712,Z 315.528,A -85,B 0,C 180,E1 -30185.052,E2 -30185.052} C_VEL
LIN {X 0,Y 36.716,Z 315.531,A -85,B 0,C 180,E1 -30190.03,E2 -30190.03} C_VEL
LIN {X 0,Y 36.722,Z 315.527,A -85,B 0,C 180,E1 -30199.955,E2 -30199.955} C_VEL
LIN {X 0,Y 36.723,Z 315.536,A -85,B 0,C 180,E1 -30204.958,E2 -30204.958} C_VEL
LIN {X 0,Y 37.132,Z 315.678,A -85,B 0,C 180,E1 -30221.862,E2 -30221.862} C_VEL
LIN {X 0,Y 37.769,Z 317.498,A -85,B 0,C 180,E1 -30225.565,E2 -30225.565} C_VEL
LIN {X 0,Y 40.015,Z 319.962,A -85,B 0,C 180,E1 -30232.431,E2 -30232.431} C_VEL
LIN {X 0,Y 41.692,Z 322.925,A -85,B 0,C 180,E1 -30237.587,E2 -30237.587} C_VEL
LIN {X 0,Y 44.392,Z 330.611,A -85,B 0,C 180,E1 -30246.817,E2 -30246.817} C_VEL
LIN {X 0,Y 46.046,Z 335.639,A -85,B 0,C 180,E1 -30251.997,E2 -30251.997} C_VEL
LIN {X 0,Y 47.705,Z 345.898,A -85,B 0,C 180,E1 -30260.478,E2 -30260.478} C_VEL
LIN {X 0,Y 49.856,Z 359.383,A -85,B 0,C 180,E1 -30271.258,E2 -30271.258} C_VEL
LIN {X 0,Y 49.858,Z 366.788,A -85,B 0,C 180,E1 -30276.967,E2 -30276.967} C_VEL
LIN {X 0,Y 49.265,Z 370.015,A -85,B 0,C 180,E1 -30279.51,E2 -30279.51} C_VEL
LIN {X 0,Y 47.849,Z 373.115,A -85,B 0,C 180,E1 -30281.994,E2 -30281.994} C_VEL
LIN {X 0,Y 41.577,Z 382.535,A -85,B 0,C 180,E1 -30291.745,E2 -30291.745} C_VEL
LIN {X 0,Y 37.795,Z 391.886,A -85,B 0,C 180,E1 -30305.266,E2 -30305.266} C_VEL
LIN {X 0,Y 36.16,Z 401.792,A -85,B 0,C 180,E1 -30324.862,E2 -30324.862} C_VEL
LIN {X 0,Y 37.605,Z 408.53,A -85,B 0,C 180,E1 -30340.771,E2 -30340.771} C_VEL
LIN {X 0,Y 38.36,Z 410.393,A -85,B 0,C 180,E1 -30345.951,E2 -30345.951} C_VEL
LIN {X 0,Y 38.934,Z 411.869,A -85,B 0,C 180,E1 -30351.163,E2 -30351.163} C_VEL
LIN {X 0,Y 43.228,Z 416.424,A -85,B 0,C 180,E1 -30370.565,E2 -30370.565} C_VEL
LIN {X 0,Y 39.773,Z 412.997,A -85,B 0,C 180,E1 -30377.984,E2 -30377.984} C_VEL
LIN {X 0,Y 34.388,Z 405.022,A -85,B 0,C 180,E1 -30395.877,E2 -30395.877} C_VEL
LIN {X 0,Y 32.252,Z 398.292,A -85,B 0,C 180,E1 -30410.597,E2 -30410.597} C_VEL
LIN {X 0,Y 32.05,Z 388.938,A -85,B 0,C 180,E1 -30429.469,E2 -30429.469} C_VEL
LIN {X 0,Y 34.84,Z 378.151,A -85,B 0,C 180,E1 -30446.995,E2 -30446.995} C_VEL
LIN {X 0,Y 40.527,Z 364.453,A -85,B 0,C 180,E1 -30462.223,E2 -30462.223} C_VEL
LIN {X 0,Y 43.058,Z 358.998,A -85,B 0,C 180,E1 -30466.626,E2 -30466.626} C_VEL
LIN {X 0,Y 43.33,Z 357.334,A -85,B 0,C 180,E1 -30468.006,E2 -30468.006} C_VEL
LIN {X 0,Y 40.784,Z 345.149,A -85,B 0,C 180,E1 -30480.303,E2 -30480.303} C_VEL
LIN {X 0,Y 39.042,Z 337.499,A -85,B 0,C 180,E1 -30488.899,E2 -30488.899} C_VEL
LIN {X 0,Y 37.382,Z 331.894,A -85,B 0,C 180,E1 -30496.408,E2 -30496.408} C_VEL
LIN {X 0,Y 36.342,Z 328.249,A -85,B 0,C 180,E1 -30501.941,E2 -30501.941} C_VEL
LIN {X 0,Y 34.811,Z 323.965,A -85,B 0,C 180,E1 -30510,E2 -30510} C_VEL
LIN {X 0,Y 33.866,Z 321.505,A -85,B 0,C 180,E1 -30515.956,E2 -30515.956} C_VEL
LIN {X 0,Y 30.53,Z 319.237,A -85,B 0,C 180,E1 -30537.413,E2 -30537.413} C_VEL
LIN {X 0,Y 30.395,Z 318.977,A -85,B 0,C 180,E1 -30556.074,E2 -30556.074} C_VEL
LIN {X 0,Y 32.236,Z 321.108,A -85,B 0,C 180,E1 -30574.146,E2 -30574.146} C_VEL
LIN {X 0,Y 33.577,Z 322.288,A -85,B 0,C 180,E1 -30580.584,E2 -30580.584} C_VEL
LIN {X 0,Y 35.681,Z 325.489,A -85,B 0,C 180,E1 -30590.013,E2 -30590.013} C_VEL
LIN {X 0,Y 36.685,Z 327.374,A -85,B 0,C 180,E1 -30593.949,E2 -30593.949} C_VEL
LIN {X 0,Y 38.514,Z 333.342,A -85,B 0,C 180,E1 -30602.621,E2 -30602.621} C_VEL
LIN {X 0,Y 40.14,Z 339.642,A -85,B 0,C 180,E1 -30610.081,E2 -30610.081} C_VEL
LIN {X 0,Y 41.533,Z 351.039,A -85,B 0,C 180,E1 -30621.072,E2 -30621.072} C_VEL
LIN {X 0,Y 42.952,Z 361.268,A -85,B 0,C 180,E1 -30630.695,E2 -30630.695} C_VEL
LIN {X 0,Y 42.944,Z 374.635,A -85,B 0,C 180,E1 -30643.226,E2 -30643.226} C_VEL
LIN {X 0,Y 43.247,Z 378.926,A -85,B 0,C 180,E1 -30647.57,E2 -30647.57} C_VEL
LIN {X 0,Y 41.577,Z 382.535,A -85,B 0,C 180,E1 -30651.745,E2 -30651.745} C_VEL
LIN {X 0,Y 39.087,Z 386.409,A -85,B 0,C 180,E1 -30657.053,E2 -30657.053} C_VEL
LIN {X 0,Y 34.113,Z 391.714,A -85,B 0,C 180,E1 -30667.675,E2 -30667.675} C_VEL
LIN {X 0,Y 30.974,Z 395.61,A -85,B 0,C 180,E1 -30678.722,E2 -30678.722} C_VEL
LIN {X 0,Y 30.101,Z 398.737,A -85,B 0,C 180,E1 -30688.139,E2 -30688.139} C_VEL
LIN {X 0,Y 30.199,Z 399.859,A -85,B 0,C 180,E1 -30691.244,E2 -30691.244} C_VEL
LIN {X 0,Y 32.119,Z 405.248,A -85,B 0,C 180,E1 -30705.873,E2 -30705.873} C_VEL
LIN {X 0,Y 33.507,Z 407.869,A -85,B 0,C 180,E1 -30714.802,E2 -30714.802} C_VEL
LIN {X 0,Y 36.22,Z 410.814,A -85,B 0,C 180,E1 -30729.095,E2 -30729.095} C_VEL
LIN {X 0,Y 30.196,Z 404.112,A -85,B 0,C 180,E1 -30744.422,E2 -30744.422} C_VEL
LIN {X 0,Y 26.783,Z 397.589,A -85,B 0,C 180,E1 -30760.856,E2 -30760.856} C_VEL
LIN {X 0,Y 25.27,Z 388.355,A -85,B 0,C 180,E1 -30783.991,E2 -30783.991} C_VEL
LIN {X 0,Y 28.289,Z 375.67,A -85,B 0,C 180,E1 -30809.798,E2 -30809.798} C_VEL
LIN {X 0,Y 35.321,Z 360.556,A -85,B 0,C 180,E1 -30828.262,E2 -30828.262} C_VEL
LIN {X 0,Y 36.1,Z 358.951,A -85,B 0,C 180,E1 -30829.641,E2 -30829.641} C_VEL
LIN {X 0,Y 35.986,Z 356.473,A -85,B 0,C 180,E1 -30832.392,E2 -30832.392} C_VEL
LIN {X 0,Y 34.107,Z 345.74,A -85,B 0,C 180,E1 -30845.663,E2 -30845.663} C_VEL
LIN {X 0,Y 32.916,Z 339.487,A -85,B 0,C 180,E1 -30854.521,E2 -30854.521} C_VEL
LIN {X 0,Y 31.389,Z 332.692,A -85,B 0,C 180,E1 -30866.169,E2 -30866.169} C_VEL
LIN {X 0,Y 30.262,Z 328.124,A -85,B 0,C 180,E1 -30876.669,E2 -30876.669} C_VEL
LIN {X 0,Y 29.01,Z 326.859,A -85,B 0,C 180,E1 -30884.276,E2 -30884.276} C_VEL
LIN {X 0,Y 27.453,Z 325.664,A -85,B 0,C 180,E1 -30900.798,E2 -30900.798} C_VEL
LIN {X 0,Y 27.349,Z 325.492,A -85,B 0,C 180,E1 -30909.559,E2 -30909.559} C_VEL
LIN {X 0,Y 27.643,Z 325.943,A -85,B 0,C 180,E1 -30919.705,E2 -30919.705} C_VEL
LIN {X 0,Y 28.625,Z 327.091,A -85,B 0,C 180,E1 -30930.587,E2 -30930.587} C_VEL
LIN {X 0,Y 29.978,Z 328.747,A -85,B 0,C 180,E1 -30939.681,E2 -30939.681} C_VEL
LIN {X 0,Y 31.269,Z 330.918,A -85,B 0,C 180,E1 -30947.008,E2 -30947.008} C_VEL
LIN {X 0,Y 31.895,Z 332.403,A -85,B 0,C 180,E1 -30950.64,E2 -30950.64} C_VEL
LIN {X 0,Y 33.173,Z 338.025,A -85,B 0,C 180,E1 -30959.997,E2 -30959.997} C_VEL
LIN {X 0,Y 34.157,Z 343.277,A -85,B 0,C 180,E1 -30967.391,E2 -30967.391} C_VEL
LIN {X 0,Y 35.1,Z 354.625,A -85,B 0,C 180,E1 -30980.509,E2 -30980.509} C_VEL
LIN {X 0,Y 35.976,Z 362.3,A -85,B 0,C 180,E1 -30989.231,E2 -30989.231} C_VEL
LIN {X 0,Y 35.965,Z 376.127,A -85,B 0,C 180,E1 -31004.961,E2 -31004.961} C_VEL
LIN {X 0,Y 36.101,Z 377.859,A -85,B 0,C 180,E1 -31007.049,E2 -31007.049} C_VEL
LIN {X 0,Y 31.606,Z 388.147,A -85,B 0,C 180,E1 -31023.594,E2 -31023.594} C_VEL
LIN {X 0,Y 29.989,Z 398.094,A -85,B 0,C 180,E1 -31046.566,E2 -31046.566} C_VEL
LIN {X 0,Y 30.199,Z 399.859,A -85,B 0,C 180,E1 -31051.244,E2 -31051.244} C_VEL
LIN {X 0,Y 29.96,Z 401.033,A -85,B 0,C 180,E1 -31055.681,E2 -31055.681} C_VEL
LIN {X 0,Y 28.553,Z 401.845,A -85,B 0,C 180,E1 -31064.004,E2 -31064.004} C_VEL
LIN {X 0,Y 27.624,Z 402.451,A -85,B 0,C 180,E1 -31073.365,E2 -31073.365} C_VEL
LIN {X 0,Y 28.095,Z 403.337,A -85,B 0,C 180,E1 -31078.622,E2 -31078.622} C_VEL
LIN {X 0,Y 29.241,Z 404.665,A -85,B 0,C 180,E1 -31084.722,E2 -31084.722} C_VEL
LIN {X 0,Y 27.566,Z 403.07,A -85,B 0,C 180,E1 -31090.112,E2 -31090.112} C_VEL
LIN {X 0,Y 22.417,Z 396.708,A -85,B 0,C 180,E1 -31106.731,E2 -31106.731} C_VEL
LIN {X 0,Y 18.905,Z 387.587,A -85,B 0,C 180,E1 -31134.672,E2 -31134.672} C_VEL
LIN {X 0,Y 21.487,Z 373.967,A -85,B 0,C 180,E1 -31172.112,E2 -31172.112} C_VEL
LIN {X 0,Y 29.164,Z 358.926,A -85,B 0,C 180,E1 -31193.847,E2 -31193.847} C_VEL
LIN {X 0,Y 28.348,Z 351.953,A -85,B 0,C 180,E1 -31204.287,E2 -31204.287} C_VEL
LIN {X 0,Y 27.604,Z 345.235,A -85,B 0,C 180,E1 -31215.25,E2 -31215.25} C_VEL
LIN {X 0,Y 26.809,Z 339.522,A -85,B 0,C 180,E1 -31226.529,E2 -31226.529} C_VEL
LIN {X 0,Y 26.48,Z 336.256,A -85,B 0,C 180,E1 -31233.805,E2 -31233.805} C_VEL
LIN {X 0,Y 26.317,Z 334.792,A -85,B 0,C 180,E1 -31237.674,E2 -31237.674} C_VEL
LIN {X 0,Y 25.537,Z 333.07,A -85,B 0,C 180,E1 -31245.975,E2 -31245.975} C_VEL
LIN {X 0,Y 24.334,Z 331.999,A -85,B 0,C 180,E1 -31265.285,E2 -31265.285} C_VEL
LIN {X 0,Y 25.074,Z 333.129,A -85,B 0,C 180,E1 -31287.234,E2 -31287.234} C_VEL
LIN {X 0,Y 26.02,Z 334.47,A -85,B 0,C 180,E1 -31296.418,E2 -31296.418} C_VEL
LIN {X 0,Y 27.061,Z 336.779,A -85,B 0,C 180,E1 -31304.943,E2 -31304.943} C_VEL
LIN {X 0,Y 27.77,Z 342.491,A -85,B 0,C 180,E1 -31316.545,E2 -31316.545} C_VEL
LIN {X 0,Y 28.141,Z 346.09,A -85,B 0,C 180,E1 -31322.587,E2 -31322.587} C_VEL
LIN {X 0,Y 28.462,Z 356.761,A -85,B 0,C 180,E1 -31337.975,E2 -31337.975} C_VEL
LIN {X 0,Y 29.029,Z 363.082,A -85,B 0,C 180,E1 -31346.993,E2 -31346.993} C_VEL
LIN {X 0,Y 28.862,Z 375.972,A -85,B 0,C 180,E1 -31365.324,E2 -31365.324} C_VEL
LIN {X 0,Y 28.719,Z 377.211,A -85,B 0,C 180,E1 -31367.231,E2 -31367.231} C_VEL
LIN {X 0,Y 24.476,Z 387.276,A -85,B 0,C 180,E1 -31388.715,E2 -31388.715} C_VEL
LIN {X 0,Y 24.186,Z 395.832,A -85,B 0,C 180,E1 -31414.165,E2 -31414.165} C_VEL
LIN {X 0,Y 27.028,Z 401.865,A -85,B 0,C 180,E1 -31432.957,E2 -31432.957} C_VEL
LIN {X 0,Y 28.095,Z 403.337,A -85,B 0,C 180,E1 -31438.622,E2 -31438.622} C_VEL
LIN {X 0,Y 28.061,Z 403.452,A -85,B 0,C 180,E1 -31441.082,E2 -31441.082} C_VEL
LIN {X 0,Y 26.962,Z 402.553,A -85,B 0,C 180,E1 -31444.908,E2 -31444.908} C_VEL
LIN {X 0,Y 24.714,Z 400.414,A -85,B 0,C 180,E1 -31448.865,E2 -31448.865} C_VEL
LIN {X 0,Y 16.377,Z 391.378,A -85,B 0,C 180,E1 -31460.424,E2 -31460.424} C_VEL
LIN {X 0,Y 15.068,Z 389.542,A -85,B 0,C 180,E1 -31465.834,E2 -31465.834} C_VEL
LIN {X 0,Y 12.638,Z 377.861,A -85,B 0,C 180,E1 -31516.152,E2 -31516.152} C_VEL
LIN {X 0,Y 17.5,Z 366.839,A -85,B 0,C 180,E1 -31548.859,E2 -31548.859} C_VEL
LIN {X 0,Y 21.862,Z 359.677,A -85,B 0,C 180,E1 -31559.509,E2 -31559.509} C_VEL
LIN {X 0,Y 22.286,Z 357.871,A -85,B 0,C 180,E1 -31562.373,E2 -31562.373} C_VEL
LIN {X 0,Y 21.955,Z 349.398,A -85,B 0,C 180,E1 -31579.86,E2 -31579.86} C_VEL
LIN {X 0,Y 21.882,Z 343.914,A -85,B 0,C 180,E1 -31592.955,E2 -31592.955} C_VEL
LIN {X 0,Y 22.054,Z 340.665,A -85,B 0,C 180,E1 -31601.804,E2 -31601.804} C_VEL
LIN {X 0,Y 21.849,Z 339.151,A -85,B 0,C 180,E1 -31608.765,E2 -31608.765} C_VEL
LIN {X 0,Y 20.995,Z 338.701,A -85,B 0,C 180,E1 -31632.03,E2 -31632.03} C_VEL
LIN {X 0,Y 21.138,Z 338.942,A -85,B 0,C 180,E1 -31638.315,E2 -31638.315} C_VEL
LIN {X 0,Y 22.084,Z 340.247,A -85,B 0,C 180,E1 -31652.892,E2 -31652.892} C_VEL
LIN {X 0,Y 22.407,Z 342.708,A -85,B 0,C 180,E1 -31661.716,E2 -31661.716} C_VEL
LIN {X 0,Y 22.443,Z 347.61,A -85,B 0,C 180,E1 -31673.252,E2 -31673.252} C_VEL
LIN {X 0,Y 21.866,Z 357.83,A -85,B 0,C 180,E1 -31692.241,E2 -31692.241} C_VEL
LIN {X 0,Y 22.122,Z 363.7,A -85,B 0,C 180,E1 -31703.393,E2 -31703.393} C_VEL
LIN {X 0,Y 21.717,Z 375.298,A -85,B 0,C 180,E1 -31725.284,E2 -31725.284} C_VEL
LIN {X 0,Y 18.326,Z 383.411,A -85,B 0,C 180,E1 -31747.448,E2 -31747.448} C_VEL
LIN {X 0,Y 18.545,Z 392.074,A -85,B 0,C 180,E1 -31780.922,E2 -31780.922} C_VEL
LIN {X 0,Y 21.633,Z 397.146,A -85,B 0,C 180,E1 -31799.164,E2 -31799.164} C_VEL
LIN {X 0,Y 21.236,Z 396.944,A -85,B 0,C 180,E1 -31804.314,E2 -31804.314} C_VEL
LIN {X 0,Y 16.301,Z 391.322,A -85,B 0,C 180,E1 -31819.715,E2 -31819.715} C_VEL
LIN {X 0,Y 15.068,Z 389.542,A -85,B 0,C 180,E1 -31825.834,E2 -31825.834} C_VEL
LIN {X 0,Y 13.449,Z 386.825,A -85,B 0,C 180,E1 -31835.153,E2 -31835.153} C_VEL
LIN {X 0,Y 11.119,Z 382.439,A -85,B 0,C 180,E1 -31850.083,E2 -31850.083} C_VEL
LIN {X 0,Y 8.763,Z 371.467,A -85,B 0,C 180,E1 -31900.107,E2 -31900.107} C_VEL
LIN {X 0,Y 10.594,Z 366.656,A -85,B 0,C 180,E1 -31918.817,E2 -31918.817} C_VEL
LIN {X 0,Y 11.587,Z 365.076,A -85,B 0,C 180,E1 -31922.78,E2 -31922.78} C_VEL
LIN {X 0,Y 15.788,Z 359.072,A -85,B 0,C 180,E1 -31931.76,E2 -31931.76} C_VEL
LIN {X 0,Y 16.509,Z 352.535,A -85,B 0,C 180,E1 -31950.001,E2 -31950.001} C_VEL
LIN {X 0,Y 17.182,Z 348.706,A -85,B 0,C 180,E1 -31961.357,E2 -31961.357} C_VEL
LIN {X 0,Y 17.966,Z 345.269,A -85,B 0,C 180,E1 -31973.029,E2 -31973.029} C_VEL
LIN {X 0,Y 17.537,Z 345.06,A -85,B 0,C 180,E1 -31986.718,E2 -31986.718} C_VEL
LIN {X 0,Y 17.777,Z 345.55,A -85,B 0,C 180,E1 -32002.25,E2 -32002.25} C_VEL
LIN {X 0,Y 17.988,Z 346.53,A -85,B 0,C 180,E1 -32010.137,E2 -32010.137} C_VEL
LIN {X 0,Y 17.151,Z 350.891,A -85,B 0,C 180,E1 -32022.674,E2 -32022.674} C_VEL
LIN {X 0,Y 15.308,Z 361.728,A -85,B 0,C 180,E1 -32049.917,E2 -32049.917} C_VEL
LIN {X 0,Y 15.288,Z 364.447,A -85,B 0,C 180,E1 -32057.339,E2 -32057.339} C_VEL
LIN {X 0,Y 14.547,Z 373.873,A -85,B 0,C 180,E1 -32083.557,E2 -32083.557} C_VEL
LIN {X 0,Y 11.867,Z 380.833,A -85,B 0,C 180,E1 -32112.775,E2 -32112.775} C_VEL
LIN {X 0,Y 13.364,Z 388.068,A -85,B 0,C 180,E1 -32152.481,E2 -32152.481} C_VEL
LIN {X 0,Y 12.15,Z 387.084,A -85,B 0,C 180,E1 -32160.274,E2 -32160.274} C_VEL
LIN {X 0,Y 5.876,Z 376.841,A -85,B 0,C 180,E1 -32220.017,E2 -32220.017} C_VEL
LIN {X 0,Y 11.587,Z 365.076,A -85,B 0,C 180,E1 -32282.78,E2 -32282.78} C_VEL
LIN {X 0,Y 10.685,Z 364.959,A -85,B 0,C 180,E1 -32285.747,E2 -32285.747} C_VEL
LIN {X 0,Y 8.71,Z 365.864,A -85,B 0,C 180,E1 -32288.332,E2 -32288.332} C_VEL
LIN {X 0,Y 2.195,Z 370.355,A -85,B 0,C 180,E1 -32295.847,E2 -32295.847} C_VEL
LIN {X 0,Y 5.356,Z 376.426,A -85,B 0,C 180,E1 -32474.413,E2 -32474.413} C_VEL
LIN {X 0,Y 5.74,Z 376.986,A -85,B 0,C 180,E1 -32476.988,E2 -32476.988} C_VEL
LIN {X 0,Y 3.525,Z 375.604,A -85,B 0,C 180,E1 -32485.044,E2 -32485.044} C_VEL
LIN {X 0,Y 7.081,Z 363.63,A -85,B 0,C 180,E1 -32316.931,E2 -32316.931} C_VEL
LIN {X 0,Y 10.602,Z 359.101,A -85,B 0,C 180,E1 -32316.007,E2 -32316.007} C_VEL
LIN {X 0,Y 12.785,Z 353.709,A -85,B 0,C 180,E1 -32334.791,E2 -32334.791} C_VEL
LIN {X 0,Y 13.651,Z 351.941,A -85,B 0,C 180,E1 -32340.989,E2 -32340.989} C_VEL
LIN {X 0,Y 13.912,Z 351.619,A -85,B 0,C 180,E1 -32357.016,E2 -32357.016} C_VEL
LIN {X 0,Y 12.441,Z 354.695,A -85,B 0,C 180,E1 -32365.596,E2 -32365.596} C_VEL
LIN {X 0,Y 8.914,Z 364.52,A -85,B 0,C 180,E1 -32399.989,E2 -32399.989} C_VEL
LIN {X 0,Y 7.659,Z 369.543,A -85,B 0,C 180,E1 -32423.412,E2 -32423.412} C_VEL
LIN {X 0,Y 7.229,Z 373.045,A -85,B 0,C 180,E1 -32443.179,E2 -32443.179} C_VEL
LIN {X 0,Y 5.74,Z 376.986,A -85,B 0,C 180,E1 -32476.988,E2 -32476.988} C_VEL
LIN {X 0,Y 5.722,Z 378.427,A -85,B 0,C 180,E1 -32483.122,E2 -32483.122} C_VEL
LIN {X 0,Y 5.722,Z 600,A -85,B 0,C 180,E1 -32483.122,E2 -32483.122} C_VEL
LIN {X 0,Y 5.722,Z 600,A -85,B 0,C 180,E1 -32483.122,E2 -32483.122}

QRS_NEXT_CUT()

QRS_NEXT()
QRS_HOME()

END
